RoboDK station: kr30 cnc 070119 curve 7 axis test 4.rdk

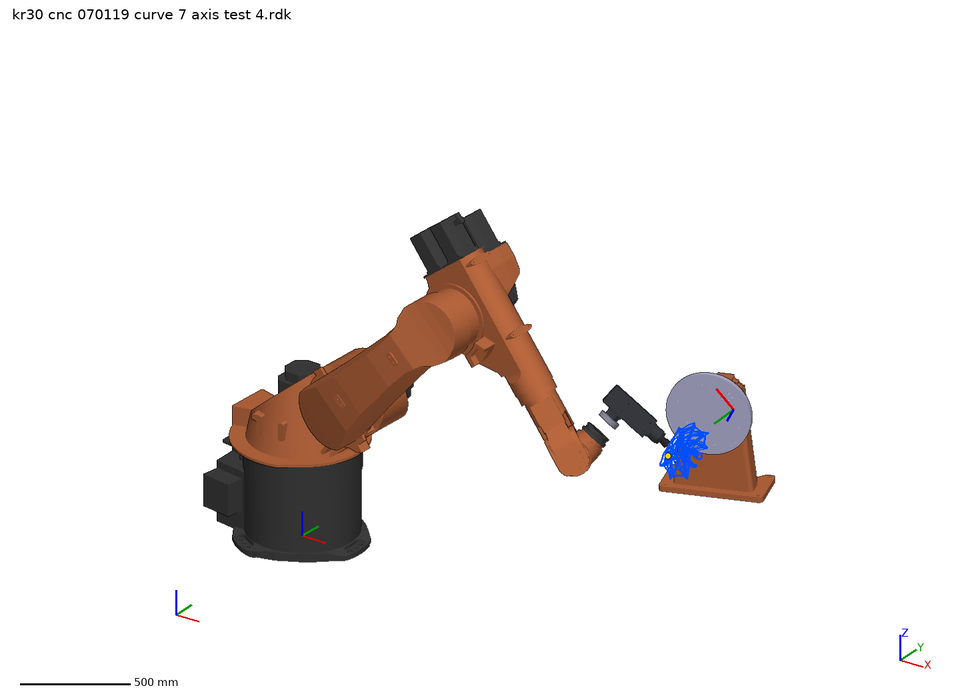
[picture v0: the station drawn from its stored meshes, robots at their saved joint values, targets as dots, program paths as lines]
Station kr30 cnc 070119 curve 7 axis test 4. Poses are relative to the parent item; angles as X-Y-Z fixed-axis rotations.
  - machining project Curve settings: C:/Temp/temp3/RhinoProject.stl | rotZ(0) | rotX(0)*rotY(0) | rotz(0) | onStart | onPathStart | onApproach | onPoint | onRetract | onFinish | onPathFinish | M_RunCode(%1)
  - frame KUKA KP1 MD250 Base at (0, 1000, 0) mm
    - robot KUKA KP1 MD250: 1 axes, payload 250 kg
        modified DH rows (alpha deg, a mm, theta deg, d mm): 0, 0, 0, 0
        base shift (1750, 1710, 820) mm, rotated rx 0 ry 90 rz -70 deg
        joint limits [-3600] to [3600]; home [0]; saved at [-138.652]
      - frame Reference Rhino at (0, -250, 250) mm
        - object RhinoPart at (0, 0, 0) mm
  - frame KUKA KR 30 HA Base at (0, 2000, 0) mm
    - robot KUKA KR 30 HA: 6 axes, payload 30 kg, reach 2033 mm, repeatability 0.05 mm, weight 665 kg
        modified DH rows (alpha deg, a mm, theta deg, d mm): 0, 0, 0, 815; -90, 350, 0, 0; 0, 850, -90, 0; -90, 145, 0, 820; 90, 0, 0, 0; -90, 0, 180, 170
        joint limits [-185, -135, -120, -350, -119, -350] to [185, 35, 158, 350, 119, 350]; home [0, -90, 90, 0, 0, 0]; saved at [2.992, -45.506, 98.07, 220.703, 109.004, -186.689]
      - tool 1/2" End Mill TCP, TCP at (337.71, -2.2, 160.57) mm, rotated rx 0 ry 90 rz 0 deg, size 415.8 x 102 x 153.6 mm
  - machining project RhinoPart Settings: rotZ(0) | rotX(90)*rotY(-155) | rotz(0) | onStart | onPathStart | onApproach | onPoint | onRetract | onFinish | onPathFinish | M_RunCode(%1)
  - program RhinoPart (1340 instructions, listed below)
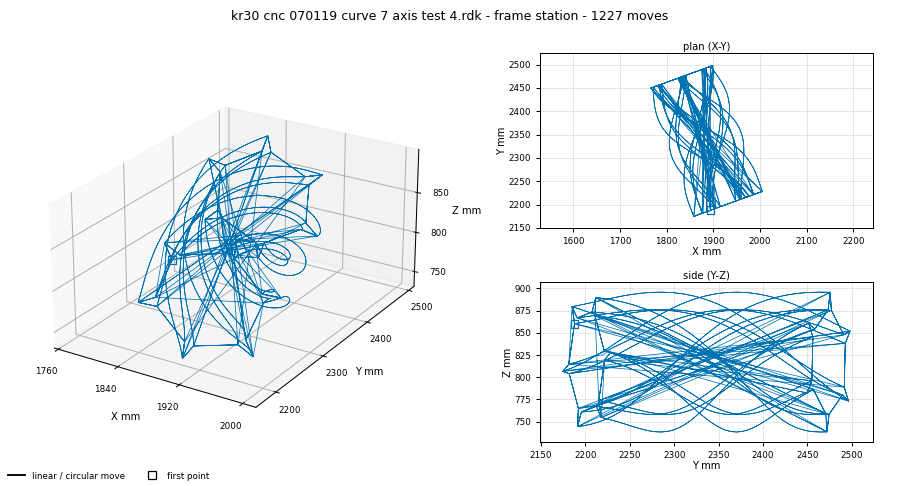
[picture p0: tool path of kr30 cnc 070119 curve 7 axis test 4.rdk in frame station, 1227 of 1227 moves have a stored position in this frame; points joined in program order, loops and branches not executed]

--- program RhinoPart (robot KUKA KR 30 HA) ---
  Set Ref.: Reference Rhino
  Set Tool: 1/2" End Mill TCP
  Show 1/2" End Mill TCP
  Set speed (1000.0 mm/s)
  MoveJ 1 to (58.93, 255.88, 290) mm, rotated rx -90 ry -25 rz 145.69 deg; joints [2.992, -45.858, 98.042, 220.619, 108.716, -186.951, -185.694]
  MoveL 2 to (58.93, 255.88, 290) mm, rotated rx -90 ry -25 rz 145.69 deg; joints [2.992, -45.858, 98.042, 220.619, 108.716, -186.951, -185.694]
  MoveL 3 to (58.93, 255.88, 290) mm, rotated rx -90 ry -25 rz 145.69 deg; joints [2.992, -45.858, 98.042, 220.619, 108.716, -186.951, -185.694]
  Set speed (60.0 mm/s)
  MoveL 4 to (37.11, 300.24, 290) mm, rotated rx -90 ry -25 rz -166.45 deg; joints [2.992, -46.004, 98.028, 220.584, 108.594, -187.061, -233.547]
  MoveL 5 to (-37.11, 208.63, 290) mm, rotated rx -90 ry -25 rz 8.11 deg; joints [2.992, -45.692, 98.056, 220.659, 108.852, -186.827, -408.107]
  Set speed (60.0 mm/s)
  MoveL 6 to (-58.93, 252.99, 290) mm, rotated rx -90 ry -25 rz -42.9 deg; joints [2.992, -45.848, 98.043, 220.621, 108.724, -186.944, -357.096]
  MoveL 7 to (21.11, 199.39, 290) mm, rotated rx -90 ry -25 rz 72.64 deg; joints [2.992, -45.658, 98.059, 220.667, 108.88, -186.802, -472.645]
  Set speed (60.0 mm/s)
  MoveL 8 to (34.79, 183.72, 290) mm, rotated rx -90 ry -25 rz 77.69 deg; joints [2.992, -46.56, 97.967, 220.451, 108.125, -187.483, -477.692]
  MoveL 9 to (21.11, 199.39, 290) mm, rotated rx -90 ry -25 rz 72.64 deg; joints [2.992, -45.658, 98.059, 220.667, 108.88, -186.802, -472.645]
  Set speed (60.0 mm/s)
  MoveL 10 to (-28.22, 202.67, 290) mm, rotated rx -90 ry -25 rz 19.2 deg; joints [2.992, -45.67, 98.058, 220.664, 108.87, -186.811, -419.196]
  MoveL 11 to (-43.85, 188.95, 290) mm, rotated rx -90 ry -25 rz 14.31 deg; joints [2.992, -46.574, 97.966, 220.447, 108.114, -187.494, -414.314]
  Set speed (60.0 mm/s)
  MoveL 12 to (-28.22, 202.67, 290) mm, rotated rx -90 ry -25 rz 19.2 deg; joints [2.992, -45.67, 98.058, 220.664, 108.87, -186.811, -419.196]
  MoveL 13 to (-43.85, 188.95, 290) mm, rotated rx -90 ry -25 rz 14.31 deg; joints [2.992, -46.574, 97.966, 220.447, 108.114, -187.494, -414.314]
  Set speed (60.0 mm/s)
  MoveL 14 to (-37.11, 208.63, 290) mm, rotated rx -90 ry -25 rz 8.11 deg; joints [2.992, -45.692, 98.056, 220.659, 108.852, -186.827, -408.107]
  MoveL 15 to (-78.63, 259.66, 290) mm, rotated rx -90 ry -25 rz -47.01 deg; joints [2.992, -46.754, 97.943, 220.404, 107.959, -187.632, -352.994]
  Set speed (60.0 mm/s)
  MoveL 16 to (-58.93, 252.99, 290) mm, rotated rx -90 ry -25 rz -42.9 deg; joints [2.992, -45.848, 98.043, 220.621, 108.724, -186.944, -357.096]
  MoveL 17 to (-78.63, 259.66, 290) mm, rotated rx -90 ry -25 rz -47.01 deg; joints [2.992, -46.754, 97.943, 220.404, 107.959, -187.632, -352.994]
  Set speed (60.0 mm/s)
  MoveL 18 to (-58.22, 263.67, 290) mm, rotated rx -90 ry -25 rz -53.21 deg; joints [2.992, -45.884, 98.039, 220.612, 108.694, -186.971, -346.787]
  MoveL 19 to (-30.72, 304.75, 290) mm, rotated rx -90 ry -25 rz -100.71 deg; joints [2.992, -46.018, 98.027, 220.58, 108.582, -187.072, -299.294]
  Set speed (60.0 mm/s)
  MoveL 20 to (-58.22, 263.67, 290) mm, rotated rx -90 ry -25 rz -53.21 deg; joints [2.992, -45.884, 98.039, 220.612, 108.694, -186.971, -346.787]
  MoveL 21 to (-30.72, 304.75, 290) mm, rotated rx -90 ry -25 rz -100.71 deg; joints [2.992, -46.018, 98.027, 220.58, 108.582, -187.072, -299.294]
  Set speed (60.0 mm/s)
  MoveL 22 to (-34.79, 325.15, 290) mm, rotated rx -90 ry -25 rz -105.16 deg; joints [2.992, -46.913, 97.922, 220.367, 107.822, -187.755, -294.84]
  MoveL 23 to (-21.11, 309.47, 290) mm, rotated rx -90 ry -25 rz -110.46 deg; joints [2.992, -46.033, 98.025, 220.576, 108.57, -187.083, -289.544]
  Set speed (60.0 mm/s)
  MoveL 24 to (-34.79, 325.15, 290) mm, rotated rx -90 ry -25 rz -105.16 deg; joints [2.992, -46.913, 97.922, 220.367, 107.822, -187.755, -294.84]
  MoveL 25 to (-21.11, 309.47, 290) mm, rotated rx -90 ry -25 rz -110.46 deg; joints [2.992, -46.033, 98.025, 220.576, 108.57, -187.083, -289.544]
  Set speed (60.0 mm/s)
  MoveL 26 to (28.22, 306.19, 290) mm, rotated rx -90 ry -25 rz -156.66 deg; joints [2.992, -46.023, 98.026, 220.579, 108.578, -187.075, -243.337]
  MoveL 27 to (43.85, 319.91, 290) mm, rotated rx -90 ry -25 rz -162.09 deg; joints [2.992, -46.901, 97.924, 220.37, 107.832, -187.745, -237.907]
  Set speed (60.0 mm/s)
  MoveL 28 to (28.22, 306.19, 290) mm, rotated rx -90 ry -25 rz -156.66 deg; joints [2.992, -46.023, 98.026, 220.579, 108.578, -187.075, -243.337]
  MoveL 29 to (43.85, 319.91, 290) mm, rotated rx -90 ry -25 rz -162.09 deg; joints [2.992, -46.901, 97.924, 220.37, 107.832, -187.745, -237.907]
  Set speed (60.0 mm/s)
  MoveL 30 to (37.11, 300.24, 290) mm, rotated rx -90 ry -25 rz -166.45 deg; joints [2.992, -46.004, 98.028, 220.584, 108.594, -187.061, -233.547]
  MoveL 31 to (78.63, 249.2, 290) mm, rotated rx -90 ry -25 rz 139.42 deg; joints [2.992, -46.728, 97.946, 220.411, 107.981, -187.612, -179.419]
  Set speed (60.0 mm/s)
  MoveL 32 to (58.93, 255.88, 290) mm, rotated rx -90 ry -25 rz 145.69 deg; joints [2.992, -45.858, 98.042, 220.619, 108.716, -186.951, -185.694]
  MoveL 33 to (78.63, 249.2, 290) mm, rotated rx -90 ry -25 rz 139.42 deg; joints [2.992, -46.728, 97.946, 220.411, 107.981, -187.612, -179.419]
  Set speed (60.0 mm/s)
  MoveL 34 to (58.22, 245.2, 290) mm, rotated rx -90 ry -25 rz 135.28 deg; joints [2.992, -45.821, 98.045, 220.627, 108.746, -186.924, -175.284]
  MoveL 35 to (30.72, 204.12, 290) mm, rotated rx -90 ry -25 rz 83.8 deg; joints [2.992, -45.676, 98.058, 220.663, 108.866, -186.815, -123.801]
  Set speed (60.0 mm/s)
  MoveL 36 to (58.22, 245.2, 290) mm, rotated rx -90 ry -25 rz 135.28 deg; joints [2.992, -45.821, 98.045, 220.627, 108.746, -186.924, -175.284]
  MoveL 37 to (30.72, 204.12, 290) mm, rotated rx -90 ry -25 rz 83.8 deg; joints [2.992, -45.676, 98.058, 220.663, 108.866, -186.815, -123.801]
  Set speed (60.0 mm/s)
  MoveL 38 to (34.79, 183.72, 290) mm, rotated rx -90 ry -25 rz 77.69 deg; joints [2.992, -46.56, 97.967, 220.451, 108.125, -187.483, -117.692]
  MoveL 39 to (-37.62, 299.82, 0) mm, rotated rx -90 ry -25 rz -92.94 deg; joints [-7.468, -50.311, 106.419, 214.538, 108.079, -179.325, 52.939]
  Set speed (60.0 mm/s)
  MoveL 40 to (10.16, 312.5, 0) mm, rotated rx -90 ry -25 rz -139.23 deg; joints [-7.468, -50.355, 106.415, 214.529, 108.039, -179.354, 99.233]
  MoveL 41 to (-37.62, 299.82, 0) mm, rotated rx -90 ry -25 rz -92.94 deg; joints [-7.468, -50.311, 106.419, 214.538, 108.079, -179.325, 52.939]
  Set speed (60.0 mm/s)
  MoveL 42 to (-55.59, 310.29, 0) mm, rotated rx -90 ry -25 rz -87.32 deg; joints [-7.468, -51.259, 106.317, 214.349, 107.213, -179.948, 47.319]
  MoveL 43 to (-45.21, 292.27, 0) mm, rotated rx -90 ry -25 rz -83.07 deg; joints [-7.468, -50.285, 106.421, 214.543, 108.102, -179.308, 43.073]
  Set speed (60.0 mm/s)
  MoveL 44 to (-55.59, 310.29, 0) mm, rotated rx -90 ry -25 rz -87.32 deg; joints [-7.468, -51.259, 106.317, 214.349, 107.213, -179.948, 47.319]
  MoveL 45 to (-45.21, 292.27, 0) mm, rotated rx -90 ry -25 rz -83.07 deg; joints [-7.468, -50.285, 106.421, 214.543, 108.102, -179.308, 43.073]
  Set speed (60.0 mm/s)
  MoveL 46 to (-58.12, 244.54, 0) mm, rotated rx -90 ry -25 rz -34.64 deg; joints [-7.468, -50.113, 106.436, 214.578, 108.256, -179.196, -5.364]
  MoveL 47 to (-76.17, 234.21, 0) mm, rotated rx -90 ry -25 rz -28.29 deg; joints [-7.468, -51.057, 106.341, 214.389, 107.4, -179.814, -11.709]
  Set speed (60.0 mm/s)
  MoveL 48 to (-58.12, 244.54, 0) mm, rotated rx -90 ry -25 rz -34.64 deg; joints [-7.468, -50.113, 106.436, 214.578, 108.256, -179.196, -5.364]
  MoveL 49 to (-76.17, 234.21, 0) mm, rotated rx -90 ry -25 rz -28.29 deg; joints [-7.468, -51.057, 106.341, 214.389, 107.4, -179.814, -11.709]
  Set speed (60.0 mm/s)
  MoveL 50 to (-55.37, 234.2, 0) mm, rotated rx -90 ry -25 rz -24.07 deg; joints [-7.468, -50.074, 106.439, 214.586, 108.291, -179.171, -15.929]
  MoveL 51 to (-20.49, 199.16, 0) mm, rotated rx -90 ry -25 rz 28.05 deg; joints [-7.468, -49.938, 106.45, 214.613, 108.412, -179.083, -68.047]
  Set speed (60.0 mm/s)
  MoveL 52 to (-55.37, 234.2, 0) mm, rotated rx -90 ry -25 rz -24.07 deg; joints [-7.468, -50.074, 106.439, 214.586, 108.291, -179.171, -15.929]
  MoveL 53 to (-20.49, 199.16, 0) mm, rotated rx -90 ry -25 rz 28.05 deg; joints [-7.468, -49.938, 106.45, 214.613, 108.412, -179.083, -68.047]
  Set speed (60.0 mm/s)
  MoveL 54 to (-20.57, 178.36, 0) mm, rotated rx -90 ry -25 rz 33.98 deg; joints [-7.468, -50.9, 106.359, 214.42, 107.545, -179.71, -73.977]
  MoveL 55 to (-10.16, 196.36, 0) mm, rotated rx -90 ry -25 rz 39.27 deg; joints [-7.468, -49.927, 106.451, 214.616, 108.422, -179.076, -79.273]
  Set speed (60.0 mm/s)
  MoveL 56 to (-20.57, 178.36, 0) mm, rotated rx -90 ry -25 rz 33.98 deg; joints [-7.468, -50.9, 106.359, 214.42, 107.545, -179.71, -73.977]
  MoveL 57 to (-10.16, 196.36, 0) mm, rotated rx -90 ry -25 rz 39.27 deg; joints [-7.468, -49.927, 106.451, 214.616, 108.422, -179.076, -79.273]
  Set speed (60.0 mm/s)
  MoveL 58 to (37.62, 209.05, 0) mm, rotated rx -90 ry -25 rz 92.57 deg; joints [-7.468, -49.977, 106.447, 214.605, 108.377, -179.109, -132.574]
  MoveL 59 to (55.59, 198.58, 0) mm, rotated rx -90 ry -25 rz 97.23 deg; joints [-7.468, -50.957, 106.353, 214.408, 107.492, -179.748, -137.234]
  Set speed (60.0 mm/s)
  MoveL 60 to (37.62, 209.05, 0) mm, rotated rx -90 ry -25 rz 92.57 deg; joints [-7.468, -49.977, 106.447, 214.605, 108.377, -179.109, -132.574]
  MoveL 61 to (55.59, 198.58, 0) mm, rotated rx -90 ry -25 rz 97.23 deg; joints [-7.468, -50.957, 106.353, 214.408, 107.492, -179.748, -137.234]
  Set speed (60.0 mm/s)
  MoveL 62 to (45.21, 216.6, 0) mm, rotated rx -90 ry -25 rz 103.54 deg; joints [-7.468, -50.007, 106.445, 214.599, 108.351, -179.128, -143.543]
  MoveL 63 to (58.12, 264.32, 0) mm, rotated rx -90 ry -25 rz 153.85 deg; joints [-7.468, -50.186, 106.43, 214.563, 108.191, -179.243, -193.845]
  Set speed (60.0 mm/s)
  MoveL 64 to (45.21, 216.6, 0) mm, rotated rx -90 ry -25 rz 103.54 deg; joints [-7.468, -50.007, 106.445, 214.599, 108.351, -179.128, -143.543]
  MoveL 65 to (58.12, 264.32, 0) mm, rotated rx -90 ry -25 rz 153.85 deg; joints [-7.468, -50.186, 106.43, 214.563, 108.191, -179.243, -193.845]
  Set speed (60.0 mm/s)
  MoveL 66 to (76.17, 274.65, 0) mm, rotated rx -90 ry -25 rz 157.93 deg; joints [-7.468, -51.166, 106.328, 214.367, 107.299, -179.886, -197.935]
  MoveL 67 to (55.37, 274.67, 0) mm, rotated rx -90 ry -25 rz 164.01 deg; joints [-7.468, -50.223, 106.427, 214.556, 108.158, -179.268, -204.014]
  Set speed (60.0 mm/s)
  MoveL 68 to (76.17, 274.65, 0) mm, rotated rx -90 ry -25 rz 157.93 deg; joints [-7.468, -51.166, 106.328, 214.367, 107.299, -179.886, -197.935]
  MoveL 69 to (55.37, 274.67, 0) mm, rotated rx -90 ry -25 rz 164.01 deg; joints [-7.468, -50.223, 106.427, 214.556, 108.158, -179.268, -204.014]
  Set speed (60.0 mm/s)
  MoveL 70 to (20.49, 309.71, 0) mm, rotated rx -90 ry -25 rz -148.94 deg; joints [-7.468, -50.346, 106.416, 214.531, 108.048, -179.347, -251.057]
  MoveL 71 to (20.57, 330.51, 0) mm, rotated rx -90 ry -25 rz -144.34 deg; joints [-7.468, -51.311, 106.31, 214.338, 107.164, -179.983, -255.665]
  Set speed (60.0 mm/s)
  MoveL 72 to (20.49, 309.71, 0) mm, rotated rx -90 ry -25 rz -148.94 deg; joints [-7.468, -50.346, 106.416, 214.531, 108.048, -179.347, -251.057]
  MoveL 73 to (20.57, 330.51, 0) mm, rotated rx -90 ry -25 rz -144.34 deg; joints [-7.468, -51.311, 106.31, 214.338, 107.164, -179.983, -255.665]
  Set speed (60.0 mm/s)
  MoveL 74 to (10.16, 312.5, 0) mm, rotated rx -90 ry -25 rz -139.23 deg; joints [-7.468, -50.355, 106.415, 214.529, 108.039, -179.354, -260.767]
  MoveL 75 to (-37.62, 299.82, 0) mm, rotated rx -90 ry -25 rz -92.94 deg; joints [-7.468, -50.311, 106.419, 214.538, 108.079, -179.325, -307.061]
  Set speed (60.0 mm/s)
  MoveL 76 to (-40.85, 296.93, 10) mm, rotated rx -90 ry -25 rz -88.96 deg; joints [-7.088, -50.198, 106.219, 214.78, 108.128, -179.56, -311.039]
  MoveL 77 to (-44.15, 293.5, 20) mm, rotated rx -90 ry -25 rz -84.58 deg; joints [-6.709, -50.079, 106.012, 215.02, 108.177, -179.796, -315.425]
  MoveL 78 to (-47.39, 289.5, 30) mm, rotated rx -90 ry -25 rz -79.81 deg; joints [-6.332, -49.955, 105.8, 215.259, 108.227, -180.032, -320.19]
  MoveL 79 to (-50.45, 284.92, 40) mm, rotated rx -90 ry -25 rz -74.69 deg; joints [-5.956, -49.826, 105.582, 215.496, 108.277, -180.268, -325.308]
  MoveL 80 to (-53.21, 279.8, 50) mm, rotated rx -90 ry -25 rz -69.25 deg; joints [-5.581, -49.692, 105.357, 215.732, 108.326, -180.504, -330.751]
  MoveL 81 to (-55.55, 274.16, 60) mm, rotated rx -90 ry -25 rz -63.51 deg; joints [-5.207, -49.552, 105.127, 215.966, 108.376, -180.74, -336.493]
  MoveL 82 to (-57.35, 268.08, 70) mm, rotated rx -90 ry -25 rz -57.49 deg; joints [-4.834, -49.408, 104.89, 216.198, 108.425, -180.977, -342.507]
  MoveL 83 to (-58.51, 261.62, 80) mm, rotated rx -90 ry -25 rz -51.24 deg; joints [-4.463, -49.259, 104.647, 216.429, 108.474, -181.215, -348.765]
  MoveL 84 to (-58.95, 254.91, 90) mm, rotated rx -90 ry -25 rz -44.76 deg; joints [-4.093, -49.106, 104.398, 216.657, 108.522, -181.454, -355.24]
  MoveL 85 to (-58.6, 248.05, 100) mm, rotated rx -90 ry -25 rz -38.1 deg; joints [-3.725, -48.95, 104.143, 216.884, 108.569, -181.693, -361.902]
  MoveL 86 to (-57.44, 241.19, 110) mm, rotated rx -90 ry -25 rz -31.28 deg; joints [-3.358, -48.79, 103.881, 217.108, 108.614, -181.935, -368.721]
  MoveL 87 to (-55.46, 234.45, 120) mm, rotated rx -90 ry -25 rz -24.34 deg; joints [-2.992, -48.627, 103.613, 217.33, 108.658, -182.178, -375.664]
  MoveL 88 to (-52.68, 227.97, 130) mm, rotated rx -90 ry -25 rz -17.3 deg; joints [-2.628, -48.462, 103.339, 217.55, 108.698, -182.423, -382.696]
  MoveL 89 to (-49.15, 221.88, 140) mm, rotated rx -90 ry -25 rz -10.22 deg; joints [-2.265, -48.294, 103.059, 217.767, 108.736, -182.671, -389.78]
  MoveL 90 to (-44.94, 216.28, 150) mm, rotated rx -90 ry -25 rz -3.12 deg; joints [-1.904, -48.126, 102.771, 217.981, 108.771, -182.922, -396.877]
  MoveL 91 to (-40.17, 211.29, 160) mm, rotated rx -90 ry -25 rz 3.94 deg; joints [-1.544, -47.956, 102.478, 218.192, 108.802, -183.176, -403.944]
  MoveL 92 to (-34.94, 206.95, 170) mm, rotated rx -90 ry -25 rz 10.94 deg; joints [-1.185, -47.786, 102.178, 218.401, 108.829, -183.434, -410.939]
  MoveL 93 to (-29.38, 203.32, 180) mm, rotated rx -90 ry -25 rz 17.81 deg; joints [-0.828, -47.615, 101.871, 218.606, 108.852, -183.696, -417.814]
  MoveL 94 to (-23.62, 200.42, 190) mm, rotated rx -90 ry -25 rz 24.52 deg; joints [-0.473, -47.444, 101.557, 218.809, 108.871, -183.961, -424.525]
  MoveL 95 to (-17.8, 198.23, 200) mm, rotated rx -90 ry -25 rz 31.02 deg; joints [-0.119, -47.272, 101.237, 219.008, 108.886, -184.23, -431.023]
  MoveL 96 to (-12.04, 196.73, 210) mm, rotated rx -90 ry -25 rz 37.26 deg; joints [0.233, -47.1, 100.911, 219.204, 108.897, -184.503, -437.262]
  MoveL 97 to (-6.46, 195.84, 220) mm, rotated rx -90 ry -25 rz 43.2 deg; joints [0.584, -46.927, 100.577, 219.397, 108.905, -184.78, -443.197]
  MoveL 98 to (-1.16, 195.49, 230) mm, rotated rx -90 ry -25 rz 48.78 deg; joints [0.933, -46.752, 100.237, 219.587, 108.909, -185.06, -448.782]
  MoveL 99 to (3.78, 195.6, 240) mm, rotated rx -90 ry -25 rz 53.97 deg; joints [1.28, -46.576, 99.891, 219.774, 108.91, -185.344, -453.974]
  MoveL 100 to (8.28, 196.07, 250) mm, rotated rx -90 ry -25 rz 58.73 deg; joints [1.626, -46.398, 99.538, 219.958, 108.908, -185.631, -458.733]
  MoveL 101 to (12.3, 196.78, 260) mm, rotated rx -90 ry -25 rz 63.02 deg; joints [1.97, -46.218, 99.178, 220.139, 108.904, -185.92, -463.017]
  MoveL 102 to (15.8, 197.64, 270) mm, rotated rx -90 ry -25 rz 66.79 deg; joints [2.312, -46.035, 98.812, 220.318, 108.898, -186.212, -466.788]
  MoveL 103 to (18.74, 198.54, 280) mm, rotated rx -90 ry -25 rz 70.01 deg; joints [2.653, -45.848, 98.439, 220.494, 108.89, -186.506, -470.01]
  MoveL 104 to (21.11, 199.39, 290) mm, rotated rx -90 ry -25 rz 72.64 deg; joints [2.992, -45.658, 98.059, 220.667, 108.88, -186.802, -472.645]
  MoveL 105 to (10.16, 312.5, 0) mm, rotated rx -90 ry -25 rz -139.23 deg; joints [-7.468, -50.355, 106.415, 214.529, 108.039, -179.354, -620.767]
  Set speed (60.0 mm/s)
  MoveL 106 to (-37.62, 299.82, 0) mm, rotated rx -90 ry -25 rz -92.94 deg; joints [-7.468, -50.311, 106.419, 214.538, 108.079, -179.325, -667.061]
  MoveL 107 to (-28.22, 202.67, 290) mm, rotated rx -90 ry -25 rz 19.2 deg; joints [2.992, -45.67, 98.058, 220.664, 108.87, -186.811, -779.196]
  Set speed (60.0 mm/s)
  MoveL 108 to (21.11, 199.39, 290) mm, rotated rx -90 ry -25 rz 72.64 deg; joints [2.992, -45.658, 98.059, 220.667, 108.88, -186.802, -832.645]
  MoveL 109 to (-28.22, 202.67, 290) mm, rotated rx -90 ry -25 rz 19.2 deg; joints [2.992, -45.67, 98.058, 220.664, 108.87, -186.811, -779.196]
  Set speed (60.0 mm/s)
  MoveL 110 to (-30.4, 203.93, 280) mm, rotated rx -90 ry -25 rz 16.58 deg; joints [2.653, -45.868, 98.437, 220.489, 108.873, -186.521, -776.579]
  MoveL 111 to (-33, 205.58, 270) mm, rotated rx -90 ry -25 rz 13.39 deg; joints [2.312, -46.064, 98.809, 220.311, 108.874, -186.234, -773.391]
  MoveL 112 to (-35.92, 207.69, 260) mm, rotated rx -90 ry -25 rz 9.67 deg; joints [1.97, -46.258, 99.175, 220.13, 108.871, -185.95, -769.674]
  MoveL 113 to (-39.07, 210.28, 250) mm, rotated rx -90 ry -25 rz 5.47 deg; joints [1.626, -46.451, 99.533, 219.946, 108.865, -185.669, -765.473]
  MoveL 114 to (-42.34, 213.41, 240) mm, rotated rx -90 ry -25 rz 0.83 deg; joints [1.28, -46.642, 99.885, 219.758, 108.855, -185.392, -760.831]
  MoveL 115 to (-45.62, 217.1, 230) mm, rotated rx -90 ry -25 rz -4.21 deg; joints [0.933, -46.832, 100.231, 219.568, 108.842, -185.119, -755.794]
  MoveL 116 to (-48.8, 221.36, 220) mm, rotated rx -90 ry -25 rz -9.59 deg; joints [0.584, -47.021, 100.57, 219.375, 108.826, -184.849, -750.406]
  MoveL 117 to (-51.74, 226.19, 210) mm, rotated rx -90 ry -25 rz -15.29 deg; joints [0.233, -47.209, 100.902, 219.178, 108.806, -184.582, -744.713]
  MoveL 118 to (-54.33, 231.55, 200) mm, rotated rx -90 ry -25 rz -21.24 deg; joints [-0.119, -47.395, 101.227, 218.979, 108.783, -184.319, -738.758]
  MoveL 119 to (-56.44, 237.4, 190) mm, rotated rx -90 ry -25 rz -27.41 deg; joints [-0.473, -47.58, 101.546, 218.777, 108.756, -184.059, -732.587]
  MoveL 120 to (-57.96, 243.66, 180) mm, rotated rx -90 ry -25 rz -33.76 deg; joints [-0.828, -47.763, 101.858, 218.572, 108.727, -183.801, -726.24]
  MoveL 121 to (-58.8, 250.25, 170) mm, rotated rx -90 ry -25 rz -40.24 deg; joints [-1.185, -47.944, 102.164, 218.365, 108.694, -183.547, -719.76]
  MoveL 122 to (-58.89, 257.04, 160) mm, rotated rx -90 ry -25 rz -46.82 deg; joints [-1.544, -48.123, 102.464, 218.154, 108.66, -183.294, -713.183]
  MoveL 123 to (-58.18, 263.92, 150) mm, rotated rx -90 ry -25 rz -53.45 deg; joints [-1.904, -48.298, 102.757, 217.942, 108.623, -183.043, -706.549]
  MoveL 124 to (-56.65, 270.74, 140) mm, rotated rx -90 ry -25 rz -60.11 deg; joints [-2.265, -48.47, 103.043, 217.727, 108.585, -182.794, -699.89]
  MoveL 125 to (-54.3, 277.38, 130) mm, rotated rx -90 ry -25 rz -66.76 deg; joints [-2.628, -48.638, 103.324, 217.51, 108.546, -182.546, -693.241]
  MoveL 126 to (-51.17, 283.7, 120) mm, rotated rx -90 ry -25 rz -73.37 deg; joints [-2.992, -48.802, 103.598, 217.291, 108.506, -182.299, -686.632]
  MoveL 127 to (-47.33, 289.58, 110) mm, rotated rx -90 ry -25 rz -79.91 deg; joints [-3.358, -48.961, 103.866, 217.07, 108.466, -182.053, -680.094]
  MoveL 128 to (-42.85, 294.92, 100) mm, rotated rx -90 ry -25 rz -86.35 deg; joints [-3.725, -49.114, 104.128, 216.848, 108.426, -181.807, -673.654]
  MoveL 129 to (-37.86, 299.62, 90) mm, rotated rx -90 ry -25 rz -92.66 deg; joints [-4.093, -49.263, 104.384, 216.623, 108.386, -181.561, -667.341]
  MoveL 130 to (-32.46, 303.64, 80) mm, rotated rx -90 ry -25 rz -98.82 deg; joints [-4.463, -49.406, 104.634, 216.397, 108.346, -181.315, -661.181]
  MoveL 131 to (-26.8, 306.94, 70) mm, rotated rx -90 ry -25 rz -104.8 deg; joints [-4.834, -49.543, 104.878, 216.169, 108.307, -181.069, -655.202]
  MoveL 132 to (-21, 309.52, 60) mm, rotated rx -90 ry -25 rz -110.57 deg; joints [-5.207, -49.675, 105.115, 215.94, 108.268, -180.823, -649.431]
  MoveL 133 to (-15.19, 311.39, 50) mm, rotated rx -90 ry -25 rz -116.1 deg; joints [-5.581, -49.801, 105.347, 215.709, 108.23, -180.577, -643.896]
  MoveL 134 to (-9.5, 312.61, 40) mm, rotated rx -90 ry -25 rz -121.38 deg; joints [-5.956, -49.921, 105.573, 215.476, 108.192, -180.331, -638.624]
  MoveL 135 to (-4.03, 313.25, 30) mm, rotated rx -90 ry -25 rz -126.35 deg; joints [-6.332, -50.037, 105.793, 215.242, 108.154, -180.086, -633.645]
  MoveL 136 to (1.12, 313.37, 20) mm, rotated rx -90 ry -25 rz -131.01 deg; joints [-6.709, -50.147, 106.006, 215.006, 108.116, -179.841, -628.989]
  MoveL 137 to (5.87, 313.09, 10) mm, rotated rx -90 ry -25 rz -135.31 deg; joints [-7.088, -50.253, 106.214, 214.768, 108.078, -179.597, -624.685]
  MoveL 138 to (10.16, 312.5, 0) mm, rotated rx -90 ry -25 rz -139.23 deg; joints [-7.468, -50.355, 106.415, 214.529, 108.039, -179.354, -620.767]
  MoveL 139 to (-37.62, 299.82, 0) mm, rotated rx -90 ry -25 rz -92.94 deg; joints [-7.468, -50.311, 106.419, 214.538, 108.079, -179.325, -667.061]
  Set speed (60.0 mm/s)
  MoveL 140 to (-40.85, 296.93, 10) mm, rotated rx -90 ry -25 rz -88.96 deg; joints [-7.088, -50.198, 106.219, 214.78, 108.128, -179.56, -671.039]
  MoveL 141 to (-44.15, 293.5, 20) mm, rotated rx -90 ry -25 rz -84.58 deg; joints [-6.709, -50.079, 106.012, 215.02, 108.177, -179.796, -675.425]
  MoveL 142 to (-47.39, 289.5, 30) mm, rotated rx -90 ry -25 rz -79.81 deg; joints [-6.332, -49.955, 105.8, 215.259, 108.227, -180.032, -680.19]
  MoveL 143 to (-50.45, 284.92, 40) mm, rotated rx -90 ry -25 rz -74.69 deg; joints [-5.956, -49.826, 105.582, 215.496, 108.277, -180.268, -685.308]
  MoveL 144 to (-53.21, 279.8, 50) mm, rotated rx -90 ry -25 rz -69.25 deg; joints [-5.581, -49.692, 105.357, 215.732, 108.326, -180.504, -690.751]
  MoveL 145 to (-55.55, 274.16, 60) mm, rotated rx -90 ry -25 rz -63.51 deg; joints [-5.207, -49.552, 105.127, 215.966, 108.376, -180.74, -696.493]
  MoveL 146 to (-57.35, 268.08, 70) mm, rotated rx -90 ry -25 rz -57.49 deg; joints [-4.834, -49.408, 104.89, 216.198, 108.425, -180.977, -702.507]
  MoveL 147 to (-58.51, 261.62, 80) mm, rotated rx -90 ry -25 rz -51.24 deg; joints [-4.463, -49.259, 104.647, 216.429, 108.474, -181.215, -708.765]
  MoveL 148 to (-58.95, 254.91, 90) mm, rotated rx -90 ry -25 rz -44.76 deg; joints [-4.093, -49.106, 104.398, 216.657, 108.522, -181.454, -715.24]
  MoveL 149 to (-58.6, 248.05, 100) mm, rotated rx -90 ry -25 rz -38.1 deg; joints [-3.725, -48.95, 104.143, 216.884, 108.569, -181.693, -721.902]
  MoveL 150 to (-57.44, 241.19, 110) mm, rotated rx -90 ry -25 rz -31.28 deg; joints [-3.358, -48.79, 103.881, 217.108, 108.614, -181.935, -728.721]
  MoveL 151 to (-55.46, 234.45, 120) mm, rotated rx -90 ry -25 rz -24.34 deg; joints [-2.992, -48.627, 103.613, 217.33, 108.658, -182.178, -735.664]
  MoveL 152 to (-52.68, 227.97, 130) mm, rotated rx -90 ry -25 rz -17.3 deg; joints [-2.628, -48.462, 103.339, 217.55, 108.698, -182.423, -742.696]
  MoveL 153 to (-49.15, 221.88, 140) mm, rotated rx -90 ry -25 rz -10.22 deg; joints [-2.265, -48.294, 103.059, 217.767, 108.736, -182.671, -749.78]
  MoveL 154 to (-44.94, 216.28, 150) mm, rotated rx -90 ry -25 rz -3.12 deg; joints [-1.904, -48.126, 102.771, 217.981, 108.771, -182.922, -756.877]
  MoveL 155 to (-40.17, 211.29, 160) mm, rotated rx -90 ry -25 rz 3.94 deg; joints [-1.544, -47.956, 102.478, 218.192, 108.802, -183.176, -763.944]
  MoveL 156 to (-34.94, 206.95, 170) mm, rotated rx -90 ry -25 rz 10.94 deg; joints [-1.185, -47.786, 102.178, 218.401, 108.829, -183.434, -770.939]
  MoveL 157 to (-29.38, 203.32, 180) mm, rotated rx -90 ry -25 rz 17.81 deg; joints [-0.828, -47.615, 101.871, 218.606, 108.852, -183.696, -777.814]
  MoveL 158 to (-23.62, 200.42, 190) mm, rotated rx -90 ry -25 rz 24.52 deg; joints [-0.473, -47.444, 101.557, 218.809, 108.871, -183.961, -784.525]
  MoveL 159 to (-17.8, 198.23, 200) mm, rotated rx -90 ry -25 rz 31.02 deg; joints [-0.119, -47.272, 101.237, 219.008, 108.886, -184.23, -791.023]
  MoveL 160 to (-12.04, 196.73, 210) mm, rotated rx -90 ry -25 rz 37.26 deg; joints [0.233, -47.1, 100.911, 219.204, 108.897, -184.503, -797.262]
  MoveL 161 to (-6.46, 195.84, 220) mm, rotated rx -90 ry -25 rz 43.2 deg; joints [0.584, -46.927, 100.577, 219.397, 108.905, -184.78, -803.197]
  MoveL 162 to (-1.16, 195.49, 230) mm, rotated rx -90 ry -25 rz 48.78 deg; joints [0.933, -46.752, 100.237, 219.587, 108.909, -185.06, -808.782]
  MoveL 163 to (3.78, 195.6, 240) mm, rotated rx -90 ry -25 rz 53.97 deg; joints [1.28, -46.576, 99.891, 219.774, 108.91, -185.344, -813.974]
  MoveL 164 to (8.28, 196.07, 250) mm, rotated rx -90 ry -25 rz 58.73 deg; joints [1.626, -46.398, 99.538, 219.958, 108.908, -185.631, -818.733]
  MoveL 165 to (12.3, 196.78, 260) mm, rotated rx -90 ry -25 rz 63.02 deg; joints [1.97, -46.218, 99.178, 220.139, 108.904, -185.92, -823.017]
  MoveL 166 to (15.8, 197.64, 270) mm, rotated rx -90 ry -25 rz 66.79 deg; joints [2.312, -46.035, 98.812, 220.318, 108.898, -186.212, -826.788]
  MoveL 167 to (18.74, 198.54, 280) mm, rotated rx -90 ry -25 rz 70.01 deg; joints [2.653, -45.848, 98.439, 220.494, 108.89, -186.506, -830.01]
  MoveL 168 to (21.11, 199.39, 290) mm, rotated rx -90 ry -25 rz 72.64 deg; joints [2.992, -45.658, 98.059, 220.667, 108.88, -186.802, -832.645]
  MoveL 169 to (34.79, 183.72, 290) mm, rotated rx -90 ry -25 rz 77.69 deg; joints [2.992, -46.56, 97.967, 220.451, 108.125, -187.483, -837.692]
  Set speed (60.0 mm/s)
  MoveL 170 to (21.11, 199.39, 290) mm, rotated rx -90 ry -25 rz 72.64 deg; joints [2.992, -45.658, 98.059, 220.667, 108.88, -186.802, -832.645]
  MoveL 171 to (-55.59, 310.29, 0) mm, rotated rx -90 ry -25 rz -87.32 deg; joints [-7.468, -51.259, 106.317, 214.349, 107.213, -179.948, -672.681]
  Set speed (60.0 mm/s)
  MoveL 172 to (-37.62, 299.82, 0) mm, rotated rx -90 ry -25 rz -92.94 deg; joints [-7.468, -50.311, 106.419, 214.538, 108.079, -179.325, -667.061]
  MoveL 173 to (34.79, 183.72, 290) mm, rotated rx -90 ry -25 rz 77.69 deg; joints [2.992, -46.56, 97.967, 220.451, 108.125, -187.483, -837.692]
  Set speed (60.0 mm/s)
  MoveL 174 to (31.73, 182.3, 280) mm, rotated rx -90 ry -25 rz 75.11 deg; joints [2.653, -46.752, 98.347, 220.278, 108.131, -187.186, -835.112]
  MoveL 175 to (27.92, 180.74, 270) mm, rotated rx -90 ry -25 rz 71.96 deg; joints [2.312, -46.941, 98.72, 220.102, 108.136, -186.891, -831.958]
  MoveL 176 to (23.38, 179.17, 260) mm, rotated rx -90 ry -25 rz 68.27 deg; joints [1.97, -47.126, 99.087, 219.924, 108.139, -186.598, -828.265]
  MoveL 177 to (18.11, 177.74, 250) mm, rotated rx -90 ry -25 rz 64.07 deg; joints [1.626, -47.308, 99.447, 219.743, 108.14, -186.307, -824.071]
  MoveL 178 to (12.17, 176.57, 240) mm, rotated rx -90 ry -25 rz 59.41 deg; joints [1.28, -47.487, 99.8, 219.56, 108.139, -186.019, -819.412]
  MoveL 179 to (5.61, 175.83, 230) mm, rotated rx -90 ry -25 rz 54.33 deg; joints [0.933, -47.665, 100.147, 219.373, 108.135, -185.733, -814.325]
  MoveL 180 to (-1.49, 175.64, 220) mm, rotated rx -90 ry -25 rz 48.85 deg; joints [0.584, -47.84, 100.487, 219.184, 108.128, -185.451, -808.851]
  MoveL 181 to (-9.03, 176.15, 210) mm, rotated rx -90 ry -25 rz 43.03 deg; joints [0.233, -48.014, 100.82, 218.992, 108.118, -185.172, -803.03]
  MoveL 182 to (-16.88, 177.46, 200) mm, rotated rx -90 ry -25 rz 36.9 deg; joints [-0.119, -48.187, 101.147, 218.797, 108.104, -184.896, -796.902]
  MoveL 183 to (-24.89, 179.66, 190) mm, rotated rx -90 ry -25 rz 30.51 deg; joints [-0.473, -48.36, 101.467, 218.598, 108.086, -184.624, -790.512]
  MoveL 184 to (-32.91, 182.83, 180) mm, rotated rx -90 ry -25 rz 23.9 deg; joints [-0.828, -48.531, 101.78, 218.397, 108.064, -184.356, -783.901]
  MoveL 185 to (-40.75, 186.98, 170) mm, rotated rx -90 ry -25 rz 17.11 deg; joints [-1.185, -48.702, 102.087, 218.193, 108.039, -184.092, -777.113]
  MoveL 186 to (-48.24, 192.12, 160) mm, rotated rx -90 ry -25 rz 10.19 deg; joints [-1.544, -48.873, 102.387, 217.985, 108.009, -183.831, -770.193]
  MoveL 187 to (-55.2, 198.19, 150) mm, rotated rx -90 ry -25 rz 3.18 deg; joints [-1.904, -49.043, 102.68, 217.775, 107.975, -183.574, -763.183]
  MoveL 188 to (-61.48, 205.13, 140) mm, rotated rx -90 ry -25 rz -3.87 deg; joints [-2.265, -49.212, 102.967, 217.562, 107.937, -183.321, -756.127]
  MoveL 189 to (-66.92, 212.81, 130) mm, rotated rx -90 ry -25 rz -10.94 deg; joints [-2.628, -49.38, 103.247, 217.346, 107.896, -183.07, -749.064]
  MoveL 190 to (-71.41, 221.1, 120) mm, rotated rx -90 ry -25 rz -17.96 deg; joints [-2.992, -49.546, 103.52, 217.128, 107.851, -182.823, -742.035]
  MoveL 191 to (-74.87, 229.83, 110) mm, rotated rx -90 ry -25 rz -24.92 deg; joints [-3.358, -49.71, 103.787, 216.907, 107.804, -182.577, -735.078]
  MoveL 192 to (-77.24, 238.83, 100) mm, rotated rx -90 ry -25 rz -31.77 deg; joints [-3.725, -49.872, 104.048, 216.684, 107.755, -182.334, -728.229]
  MoveL 193 to (-78.53, 247.91, 90) mm, rotated rx -90 ry -25 rz -38.48 deg; joints [-4.093, -50.03, 104.302, 216.459, 107.704, -182.093, -721.522]
  MoveL 194 to (-78.77, 256.9, 80) mm, rotated rx -90 ry -25 rz -45.01 deg; joints [-4.463, -50.185, 104.551, 216.231, 107.651, -181.852, -714.991]
  MoveL 195 to (-78, 265.63, 70) mm, rotated rx -90 ry -25 rz -51.33 deg; joints [-4.834, -50.336, 104.793, 216.002, 107.597, -181.613, -708.666]
  MoveL 196 to (-76.35, 273.96, 60) mm, rotated rx -90 ry -25 rz -57.42 deg; joints [-5.207, -50.483, 105.028, 215.77, 107.542, -181.374, -702.579]
  MoveL 197 to (-73.92, 281.75, 50) mm, rotated rx -90 ry -25 rz -63.24 deg; joints [-5.581, -50.625, 105.258, 215.538, 107.487, -181.136, -696.759]
  MoveL 198 to (-70.87, 288.9, 40) mm, rotated rx -90 ry -25 rz -68.76 deg; joints [-5.956, -50.762, 105.482, 215.303, 107.432, -180.898, -691.235]
  MoveL 199 to (-67.34, 295.36, 30) mm, rotated rx -90 ry -25 rz -73.96 deg; joints [-6.332, -50.894, 105.7, 215.067, 107.377, -180.661, -686.036]
  MoveL 200 to (-63.51, 301.08, 20) mm, rotated rx -90 ry -25 rz -78.81 deg; joints [-6.709, -51.021, 105.911, 214.829, 107.322, -180.423, -681.192]
  MoveL 201 to (-59.54, 306.05, 10) mm, rotated rx -90 ry -25 rz -83.27 deg; joints [-7.088, -51.143, 106.117, 214.59, 107.267, -180.186, -676.73]
  MoveL 202 to (-55.59, 310.29, 0) mm, rotated rx -90 ry -25 rz -87.32 deg; joints [-7.468, -51.259, 106.317, 214.349, 107.213, -179.948, -672.681]
  MoveL 203 to (34.79, 183.72, 290) mm, rotated rx -90 ry -25 rz 77.69 deg; joints [2.992, -46.56, 97.967, 220.451, 108.125, -187.483, -837.692]
  Set speed (60.0 mm/s)
  MoveL 204 to (30.72, 204.12, 290) mm, rotated rx -90 ry -25 rz 83.8 deg; joints [2.992, -45.676, 98.058, 220.663, 108.866, -186.815, -843.801]
  MoveL 205 to (-55.59, 310.29, 0) mm, rotated rx -90 ry -25 rz -87.32 deg; joints [-7.468, -51.259, 106.317, 214.349, 107.213, -179.948, -672.681]
  Set speed (60.0 mm/s)
  MoveL 206 to (-45.21, 292.27, 0) mm, rotated rx -90 ry -25 rz -83.07 deg; joints [-7.468, -50.285, 106.421, 214.543, 108.102, -179.308, -676.927]
  MoveL 207 to (-55.59, 310.29, 0) mm, rotated rx -90 ry -25 rz -87.32 deg; joints [-7.468, -51.259, 106.317, 214.349, 107.213, -179.948, -672.681]
  Set speed (60.0 mm/s)
  MoveL 208 to (-59.54, 306.05, 10) mm, rotated rx -90 ry -25 rz -83.27 deg; joints [-7.088, -51.143, 106.117, 214.59, 107.267, -180.186, -676.73]
  MoveL 209 to (-63.51, 301.08, 20) mm, rotated rx -90 ry -25 rz -78.81 deg; joints [-6.709, -51.021, 105.911, 214.829, 107.322, -180.423, -681.192]
  MoveL 210 to (-67.34, 295.36, 30) mm, rotated rx -90 ry -25 rz -73.96 deg; joints [-6.332, -50.894, 105.7, 215.067, 107.377, -180.661, -686.036]
  MoveL 211 to (-70.87, 288.9, 40) mm, rotated rx -90 ry -25 rz -68.76 deg; joints [-5.956, -50.762, 105.482, 215.303, 107.432, -180.898, -691.235]
  MoveL 212 to (-73.92, 281.75, 50) mm, rotated rx -90 ry -25 rz -63.24 deg; joints [-5.581, -50.625, 105.258, 215.538, 107.487, -181.136, -696.759]
  MoveL 213 to (-76.35, 273.96, 60) mm, rotated rx -90 ry -25 rz -57.42 deg; joints [-5.207, -50.483, 105.028, 215.77, 107.542, -181.374, -702.579]
  MoveL 214 to (-78, 265.63, 70) mm, rotated rx -90 ry -25 rz -51.33 deg; joints [-4.834, -50.336, 104.793, 216.002, 107.597, -181.613, -708.666]
  MoveL 215 to (-78.77, 256.9, 80) mm, rotated rx -90 ry -25 rz -45.01 deg; joints [-4.463, -50.185, 104.551, 216.231, 107.651, -181.852, -714.991]
  MoveL 216 to (-78.53, 247.91, 90) mm, rotated rx -90 ry -25 rz -38.48 deg; joints [-4.093, -50.03, 104.302, 216.459, 107.704, -182.093, -721.522]
  MoveL 217 to (-77.24, 238.83, 100) mm, rotated rx -90 ry -25 rz -31.77 deg; joints [-3.725, -49.872, 104.048, 216.684, 107.755, -182.334, -728.229]
  MoveL 218 to (-74.87, 229.83, 110) mm, rotated rx -90 ry -25 rz -24.92 deg; joints [-3.358, -49.71, 103.787, 216.907, 107.804, -182.577, -735.078]
  MoveL 219 to (-71.41, 221.1, 120) mm, rotated rx -90 ry -25 rz -17.96 deg; joints [-2.992, -49.546, 103.52, 217.128, 107.851, -182.823, -742.035]
  MoveL 220 to (-66.92, 212.81, 130) mm, rotated rx -90 ry -25 rz -10.94 deg; joints [-2.628, -49.38, 103.247, 217.346, 107.896, -183.07, -749.064]
  MoveL 221 to (-61.48, 205.13, 140) mm, rotated rx -90 ry -25 rz -3.87 deg; joints [-2.265, -49.212, 102.967, 217.562, 107.937, -183.321, -756.127]
  MoveL 222 to (-55.2, 198.19, 150) mm, rotated rx -90 ry -25 rz 3.18 deg; joints [-1.904, -49.043, 102.68, 217.775, 107.975, -183.574, -763.183]
  MoveL 223 to (-48.24, 192.12, 160) mm, rotated rx -90 ry -25 rz 10.19 deg; joints [-1.544, -48.873, 102.387, 217.985, 108.009, -183.831, -770.193]
  MoveL 224 to (-40.75, 186.98, 170) mm, rotated rx -90 ry -25 rz 17.11 deg; joints [-1.185, -48.702, 102.087, 218.193, 108.039, -184.092, -777.113]
  MoveL 225 to (-32.91, 182.83, 180) mm, rotated rx -90 ry -25 rz 23.9 deg; joints [-0.828, -48.531, 101.78, 218.397, 108.064, -184.356, -783.901]
  MoveL 226 to (-24.89, 179.66, 190) mm, rotated rx -90 ry -25 rz 30.51 deg; joints [-0.473, -48.36, 101.467, 218.598, 108.086, -184.624, -790.512]
  MoveL 227 to (-16.88, 177.46, 200) mm, rotated rx -90 ry -25 rz 36.9 deg; joints [-0.119, -48.187, 101.147, 218.797, 108.104, -184.896, -796.902]
  MoveL 228 to (-9.03, 176.15, 210) mm, rotated rx -90 ry -25 rz 43.03 deg; joints [0.233, -48.014, 100.82, 218.992, 108.118, -185.172, -803.03]
  MoveL 229 to (-1.49, 175.64, 220) mm, rotated rx -90 ry -25 rz 48.85 deg; joints [0.584, -47.84, 100.487, 219.184, 108.128, -185.451, -808.851]
  MoveL 230 to (5.61, 175.83, 230) mm, rotated rx -90 ry -25 rz 54.33 deg; joints [0.933, -47.665, 100.147, 219.373, 108.135, -185.733, -814.325]
  MoveL 231 to (12.17, 176.57, 240) mm, rotated rx -90 ry -25 rz 59.41 deg; joints [1.28, -47.487, 99.8, 219.56, 108.139, -186.019, -819.412]
  MoveL 232 to (18.11, 177.74, 250) mm, rotated rx -90 ry -25 rz 64.07 deg; joints [1.626, -47.308, 99.447, 219.743, 108.14, -186.307, -824.071]
  MoveL 233 to (23.38, 179.17, 260) mm, rotated rx -90 ry -25 rz 68.27 deg; joints [1.97, -47.126, 99.087, 219.924, 108.139, -186.598, -828.265]
  MoveL 234 to (27.92, 180.74, 270) mm, rotated rx -90 ry -25 rz 71.96 deg; joints [2.312, -46.941, 98.72, 220.102, 108.136, -186.891, -831.958]
  MoveL 235 to (31.73, 182.3, 280) mm, rotated rx -90 ry -25 rz 75.11 deg; joints [2.653, -46.752, 98.347, 220.278, 108.131, -187.186, -835.112]
  MoveL 236 to (34.79, 183.72, 290) mm, rotated rx -90 ry -25 rz 77.69 deg; joints [2.992, -46.56, 97.967, 220.451, 108.125, -187.483, -837.692]
  MoveL 237 to (30.72, 204.12, 290) mm, rotated rx -90 ry -25 rz 83.8 deg; joints [2.992, -45.676, 98.058, 220.663, 108.866, -186.815, -843.801]
  Set speed (60.0 mm/s)
  MoveL 238 to (28.54, 202.85, 280) mm, rotated rx -90 ry -25 rz 81.18 deg; joints [2.653, -45.864, 98.438, 220.49, 108.877, -186.518, -841.184]
  MoveL 239 to (25.81, 201.43, 270) mm, rotated rx -90 ry -25 rz 77.98 deg; joints [2.312, -46.049, 98.811, 220.314, 108.886, -186.222, -837.983]
  MoveL 240 to (22.53, 199.96, 260) mm, rotated rx -90 ry -25 rz 74.23 deg; joints [1.97, -46.229, 99.177, 220.136, 108.895, -185.929, -834.232]
  MoveL 241 to (18.7, 198.53, 250) mm, rotated rx -90 ry -25 rz 69.97 deg; joints [1.626, -46.407, 99.537, 219.956, 108.901, -185.637, -829.967]
  MoveL 242 to (14.35, 197.26, 240) mm, rotated rx -90 ry -25 rz 65.22 deg; joints [1.28, -46.582, 99.89, 219.772, 108.905, -185.349, -825.225]
  MoveL 243 to (9.52, 196.26, 230) mm, rotated rx -90 ry -25 rz 60.04 deg; joints [0.933, -46.755, 100.237, 219.586, 108.907, -185.063, -820.042]
  MoveL 244 to (4.24, 195.64, 220) mm, rotated rx -90 ry -25 rz 54.46 deg; joints [0.584, -46.926, 100.577, 219.397, 108.906, -184.78, -814.46]
  MoveL 245 to (-1.41, 195.5, 210) mm, rotated rx -90 ry -25 rz 48.52 deg; joints [0.233, -47.095, 100.911, 219.205, 108.901, -184.5, -808.518]
  MoveL 246 to (-7.35, 195.94, 200) mm, rotated rx -90 ry -25 rz 42.26 deg; joints [-0.119, -47.264, 101.238, 219.01, 108.893, -184.224, -802.261]
  MoveL 247 to (-13.47, 197.04, 190) mm, rotated rx -90 ry -25 rz 35.73 deg; joints [-0.473, -47.431, 101.558, 218.812, 108.882, -183.952, -795.734]
  MoveL 248 to (-19.65, 198.85, 180) mm, rotated rx -90 ry -25 rz 28.98 deg; joints [-0.828, -47.598, 101.872, 218.61, 108.866, -183.684, -788.982]
  MoveL 249 to (-25.78, 201.42, 170) mm, rotated rx -90 ry -25 rz 22.05 deg; joints [-1.185, -47.765, 102.179, 218.406, 108.847, -183.419, -782.053]
  MoveL 250 to (-31.7, 204.73, 160) mm, rotated rx -90 ry -25 rz 14.99 deg; joints [-1.544, -47.932, 102.48, 218.198, 108.823, -183.159, -774.993]
  MoveL 251 to (-37.3, 208.79, 150) mm, rotated rx -90 ry -25 rz 7.85 deg; joints [-1.904, -48.098, 102.774, 217.987, 108.795, -182.902, -767.85]
  MoveL 252 to (-42.45, 213.53, 140) mm, rotated rx -90 ry -25 rz 0.67 deg; joints [-2.265, -48.263, 103.061, 217.774, 108.763, -182.649, -760.67]
  MoveL 253 to (-47.02, 218.88, 130) mm, rotated rx -90 ry -25 rz -6.5 deg; joints [-2.628, -48.428, 103.342, 217.557, 108.727, -182.399, -753.496]
  MoveL 254 to (-50.93, 224.75, 120) mm, rotated rx -90 ry -25 rz -13.63 deg; joints [-2.992, -48.591, 103.616, 217.338, 108.689, -182.153, -746.37]
  MoveL 255 to (-54.1, 231.02, 110) mm, rotated rx -90 ry -25 rz -20.67 deg; joints [-3.358, -48.752, 103.884, 217.116, 108.647, -181.909, -739.332]
  MoveL 256 to (-56.49, 237.56, 100) mm, rotated rx -90 ry -25 rz -27.58 deg; joints [-3.725, -48.911, 104.146, 216.892, 108.602, -181.667, -732.418]
  MoveL 257 to (-58.06, 244.24, 90) mm, rotated rx -90 ry -25 rz -34.34 deg; joints [-4.093, -49.068, 104.401, 216.666, 108.556, -181.427, -725.663]
  MoveL 258 to (-58.85, 250.92, 80) mm, rotated rx -90 ry -25 rz -40.9 deg; joints [-4.463, -49.221, 104.65, 216.437, 108.508, -181.189, -719.1]
  MoveL 259 to (-58.87, 257.48, 70) mm, rotated rx -90 ry -25 rz -47.24 deg; joints [-4.834, -49.37, 104.893, 216.206, 108.459, -180.952, -712.759]
  MoveL 260 to (-58.2, 263.79, 60) mm, rotated rx -90 ry -25 rz -53.33 deg; joints [-5.207, -49.515, 105.13, 215.974, 108.409, -180.716, -706.668]
  MoveL 261 to (-56.92, 269.76, 50) mm, rotated rx -90 ry -25 rz -59.14 deg; joints [-5.581, -49.656, 105.36, 215.739, 108.358, -180.48, -700.857]
  MoveL 262 to (-55.13, 275.3, 40) mm, rotated rx -90 ry -25 rz -64.65 deg; joints [-5.956, -49.792, 105.585, 215.503, 108.307, -180.245, -695.351]
  MoveL 263 to (-52.95, 280.35, 30) mm, rotated rx -90 ry -25 rz -69.82 deg; joints [-6.332, -49.923, 105.803, 215.266, 108.256, -180.01, -690.178]
  MoveL 264 to (-50.48, 284.87, 20) mm, rotated rx -90 ry -25 rz -74.63 deg; joints [-6.709, -50.049, 106.015, 215.026, 108.204, -179.776, -685.365]
  MoveL 265 to (-47.86, 288.84, 10) mm, rotated rx -90 ry -25 rz -79.06 deg; joints [-7.088, -50.169, 106.221, 214.785, 108.153, -179.542, -680.939]
  MoveL 266 to (-45.21, 292.27, 0) mm, rotated rx -90 ry -25 rz -83.07 deg; joints [-7.468, -50.285, 106.421, 214.543, 108.102, -179.308, -676.927]
  MoveL 267 to (30.72, 204.12, 290) mm, rotated rx -90 ry -25 rz 83.8 deg; joints [2.992, -45.676, 98.058, 220.663, 108.866, -186.815, -843.801]
  Set speed (60.0 mm/s)
  MoveL 268 to (58.22, 245.2, 290) mm, rotated rx -90 ry -25 rz 135.28 deg; joints [2.992, -45.821, 98.045, 220.627, 108.746, -186.924, -895.284]
  MoveL 269 to (-45.21, 292.27, 0) mm, rotated rx -90 ry -25 rz -83.07 deg; joints [-7.468, -50.285, 106.421, 214.543, 108.102, -179.308, -1036.927]
  Set speed (60.0 mm/s)
  MoveL 270 to (-58.12, 244.54, 0) mm, rotated rx -90 ry -25 rz -34.64 deg; joints [-7.468, -50.113, 106.436, 214.578, 108.256, -179.196, -1085.364]
  MoveL 271 to (-45.21, 292.27, 0) mm, rotated rx -90 ry -25 rz -83.07 deg; joints [-7.468, -50.285, 106.421, 214.543, 108.102, -179.308, -1036.927]
  Set speed (60.0 mm/s)
  MoveL 272 to (-47.86, 288.84, 10) mm, rotated rx -90 ry -25 rz -79.06 deg; joints [-7.088, -50.169, 106.221, 214.785, 108.153, -179.542, -1040.939]
  MoveL 273 to (-50.48, 284.87, 20) mm, rotated rx -90 ry -25 rz -74.63 deg; joints [-6.709, -50.049, 106.015, 215.026, 108.204, -179.776, -1045.365]
  MoveL 274 to (-52.95, 280.35, 30) mm, rotated rx -90 ry -25 rz -69.82 deg; joints [-6.332, -49.923, 105.803, 215.266, 108.256, -180.01, -1050.178]
  MoveL 275 to (-55.13, 275.3, 40) mm, rotated rx -90 ry -25 rz -64.65 deg; joints [-5.956, -49.792, 105.585, 215.503, 108.307, -180.245, -1055.351]
  MoveL 276 to (-56.92, 269.76, 50) mm, rotated rx -90 ry -25 rz -59.14 deg; joints [-5.581, -49.656, 105.36, 215.739, 108.358, -180.48, -1060.857]
  MoveL 277 to (-58.2, 263.79, 60) mm, rotated rx -90 ry -25 rz -53.33 deg; joints [-5.207, -49.515, 105.13, 215.974, 108.409, -180.716, -1066.668]
  MoveL 278 to (-58.87, 257.48, 70) mm, rotated rx -90 ry -25 rz -47.24 deg; joints [-4.834, -49.37, 104.893, 216.206, 108.459, -180.952, -1072.759]
  MoveL 279 to (-58.85, 250.92, 80) mm, rotated rx -90 ry -25 rz -40.9 deg; joints [-4.463, -49.221, 104.65, 216.437, 108.508, -181.189, -1079.1]
  MoveL 280 to (-58.06, 244.24, 90) mm, rotated rx -90 ry -25 rz -34.34 deg; joints [-4.093, -49.068, 104.401, 216.666, 108.556, -181.427, -1085.663]
  MoveL 281 to (-56.49, 237.56, 100) mm, rotated rx -90 ry -25 rz -27.58 deg; joints [-3.725, -48.911, 104.146, 216.892, 108.602, -181.667, -1092.418]
  MoveL 282 to (-54.1, 231.02, 110) mm, rotated rx -90 ry -25 rz -20.67 deg; joints [-3.358, -48.752, 103.884, 217.116, 108.647, -181.909, -1099.332]
  MoveL 283 to (-50.93, 224.75, 120) mm, rotated rx -90 ry -25 rz -13.63 deg; joints [-2.992, -48.591, 103.616, 217.338, 108.689, -182.153, -1106.37]
  MoveL 284 to (-47.02, 218.88, 130) mm, rotated rx -90 ry -25 rz -6.5 deg; joints [-2.628, -48.428, 103.342, 217.557, 108.727, -182.399, -1113.496]
  MoveL 285 to (-42.45, 213.53, 140) mm, rotated rx -90 ry -25 rz 0.67 deg; joints [-2.265, -48.263, 103.061, 217.774, 108.763, -182.649, -1120.67]
  MoveL 286 to (-37.3, 208.79, 150) mm, rotated rx -90 ry -25 rz 7.85 deg; joints [-1.904, -48.098, 102.774, 217.987, 108.795, -182.902, -1127.85]
  MoveL 287 to (-31.7, 204.73, 160) mm, rotated rx -90 ry -25 rz 14.99 deg; joints [-1.544, -47.932, 102.48, 218.198, 108.823, -183.159, -1134.993]
  MoveL 288 to (-25.78, 201.42, 170) mm, rotated rx -90 ry -25 rz 22.05 deg; joints [-1.185, -47.765, 102.179, 218.406, 108.847, -183.419, -1142.053]
  MoveL 289 to (-19.65, 198.85, 180) mm, rotated rx -90 ry -25 rz 28.98 deg; joints [-0.828, -47.598, 101.872, 218.61, 108.866, -183.684, -1148.982]
  MoveL 290 to (-13.47, 197.04, 190) mm, rotated rx -90 ry -25 rz 35.73 deg; joints [-0.473, -47.431, 101.558, 218.812, 108.882, -183.952, -1155.734]
  MoveL 291 to (-7.35, 195.94, 200) mm, rotated rx -90 ry -25 rz 42.26 deg; joints [-0.119, -47.264, 101.238, 219.01, 108.893, -184.224, -1162.261]
  MoveL 292 to (-1.41, 195.5, 210) mm, rotated rx -90 ry -25 rz 48.52 deg; joints [0.233, -47.095, 100.911, 219.205, 108.901, -184.5, -1168.518]
  MoveL 293 to (4.24, 195.64, 220) mm, rotated rx -90 ry -25 rz 54.46 deg; joints [0.584, -46.926, 100.577, 219.397, 108.906, -184.78, -1174.46]
  MoveL 294 to (9.52, 196.26, 230) mm, rotated rx -90 ry -25 rz 60.04 deg; joints [0.933, -46.755, 100.237, 219.586, 108.907, -185.063, -1180.042]
  MoveL 295 to (14.35, 197.26, 240) mm, rotated rx -90 ry -25 rz 65.22 deg; joints [1.28, -46.582, 99.89, 219.772, 108.905, -185.349, -1185.225]
  MoveL 296 to (18.7, 198.53, 250) mm, rotated rx -90 ry -25 rz 69.97 deg; joints [1.626, -46.407, 99.537, 219.956, 108.901, -185.637, -1189.967]
  MoveL 297 to (22.53, 199.96, 260) mm, rotated rx -90 ry -25 rz 74.23 deg; joints [1.97, -46.229, 99.177, 220.136, 108.895, -185.929, -1194.232]
  MoveL 298 to (25.81, 201.43, 270) mm, rotated rx -90 ry -25 rz 77.98 deg; joints [2.312, -46.049, 98.811, 220.314, 108.886, -186.222, -1197.983]
  MoveL 299 to (28.54, 202.85, 280) mm, rotated rx -90 ry -25 rz 81.18 deg; joints [2.653, -45.864, 98.438, 220.49, 108.877, -186.518, -1201.184]
  MoveL 300 to (30.72, 204.12, 290) mm, rotated rx -90 ry -25 rz 83.8 deg; joints [2.992, -45.676, 98.058, 220.663, 108.866, -186.815, -1203.801]
  MoveL 301 to (58.22, 245.2, 290) mm, rotated rx -90 ry -25 rz 135.28 deg; joints [2.992, -45.821, 98.045, 220.627, 108.746, -186.924, -1255.284]
  Set speed (60.0 mm/s)
  MoveL 302 to (57.77, 242.72, 280) mm, rotated rx -90 ry -25 rz 132.81 deg; joints [2.653, -46.006, 98.425, 220.456, 108.759, -186.624, -1252.814]
  MoveL 303 to (57.08, 239.72, 270) mm, rotated rx -90 ry -25 rz 129.79 deg; joints [2.312, -46.186, 98.799, 220.282, 108.773, -186.324, -1249.788]
  MoveL 304 to (56.08, 236.26, 260) mm, rotated rx -90 ry -25 rz 126.23 deg; joints [1.97, -46.361, 99.166, 220.105, 108.786, -186.025, -1246.235]
  MoveL 305 to (54.69, 232.42, 250) mm, rotated rx -90 ry -25 rz 122.18 deg; joints [1.626, -46.53, 99.527, 219.927, 108.798, -185.728, -1242.184]
  MoveL 306 to (52.84, 228.29, 240) mm, rotated rx -90 ry -25 rz 117.66 deg; joints [1.28, -46.696, 99.881, 219.746, 108.81, -185.432, -1237.664]
  MoveL 307 to (50.46, 223.96, 230) mm, rotated rx -90 ry -25 rz 112.71 deg; joints [0.933, -46.857, 100.229, 219.562, 108.822, -185.137, -1232.705]
  MoveL 308 to (47.51, 219.54, 220) mm, rotated rx -90 ry -25 rz 107.34 deg; joints [0.584, -47.015, 100.57, 219.376, 108.831, -184.844, -1227.337]
  MoveL 309 to (43.95, 215.15, 210) mm, rotated rx -90 ry -25 rz 101.59 deg; joints [0.233, -47.169, 100.905, 219.188, 108.84, -184.553, -1221.59]
  MoveL 310 to (39.77, 210.92, 200) mm, rotated rx -90 ry -25 rz 95.5 deg; joints [-0.119, -47.32, 101.233, 218.997, 108.846, -184.265, -1215.499]
  MoveL 311 to (34.96, 206.97, 190) mm, rotated rx -90 ry -25 rz 89.1 deg; joints [-0.473, -47.469, 101.555, 218.803, 108.85, -183.979, -1209.096]
  MoveL 312 to (29.57, 203.44, 180) mm, rotated rx -90 ry -25 rz 82.42 deg; joints [-0.828, -47.616, 101.871, 218.606, 108.852, -183.696, -1202.421]
  MoveL 313 to (23.65, 200.44, 170) mm, rotated rx -90 ry -25 rz 75.51 deg; joints [-1.185, -47.761, 102.18, 218.406, 108.85, -183.417, -1195.511]
  MoveL 314 to (17.28, 198.07, 160) mm, rotated rx -90 ry -25 rz 68.41 deg; joints [-1.544, -47.906, 102.482, 218.204, 108.844, -183.141, -1188.409]
  MoveL 315 to (10.57, 196.44, 150) mm, rotated rx -90 ry -25 rz 61.16 deg; joints [-1.904, -48.051, 102.777, 217.998, 108.835, -182.869, -1181.159]
  MoveL 316 to (3.62, 195.59, 140) mm, rotated rx -90 ry -25 rz 53.81 deg; joints [-2.265, -48.195, 103.067, 217.789, 108.821, -182.601, -1173.808]
  MoveL 317 to (-3.42, 195.58, 130) mm, rotated rx -90 ry -25 rz 46.4 deg; joints [-2.628, -48.339, 103.349, 217.577, 108.803, -182.338, -1166.404]
  MoveL 318 to (-10.42, 196.41, 120) mm, rotated rx -90 ry -25 rz 38.99 deg; joints [-2.992, -48.483, 103.625, 217.362, 108.781, -182.078, -1158.993]
  MoveL 319 to (-17.25, 198.06, 110) mm, rotated rx -90 ry -25 rz 31.62 deg; joints [-3.358, -48.627, 103.895, 217.144, 108.754, -181.823, -1151.625]
  MoveL 320 to (-23.78, 200.49, 100) mm, rotated rx -90 ry -25 rz 24.35 deg; joints [-3.725, -48.771, 104.157, 216.923, 108.724, -181.571, -1144.346]
  MoveL 321 to (-29.89, 203.62, 90) mm, rotated rx -90 ry -25 rz 17.2 deg; joints [-4.093, -48.915, 104.414, 216.699, 108.689, -181.323, -1137.203]
  MoveL 322 to (-35.48, 207.36, 80) mm, rotated rx -90 ry -25 rz 10.24 deg; joints [-4.463, -49.058, 104.664, 216.472, 108.65, -181.078, -1130.238]
  MoveL 323 to (-40.49, 211.59, 70) mm, rotated rx -90 ry -25 rz 3.49 deg; joints [-4.834, -49.199, 104.907, 216.243, 108.608, -180.837, -1123.492]
  MoveL 324 to (-44.86, 216.19, 60) mm, rotated rx -90 ry -25 rz -3 deg; joints [-5.207, -49.339, 105.145, 216.011, 108.563, -180.597, -1117.004]
  MoveL 325 to (-48.58, 221.03, 50) mm, rotated rx -90 ry -25 rz -9.19 deg; joints [-5.581, -49.477, 105.375, 215.777, 108.516, -180.36, -1110.81]
  MoveL 326 to (-51.63, 225.99, 40) mm, rotated rx -90 ry -25 rz -15.06 deg; joints [-5.956, -49.611, 105.6, 215.541, 108.466, -180.125, -1104.943]
  MoveL 327 to (-54.06, 230.92, 30) mm, rotated rx -90 ry -25 rz -20.56 deg; joints [-6.332, -49.743, 105.818, 215.303, 108.415, -179.891, -1099.435]
  MoveL 328 to (-55.91, 235.73, 20) mm, rotated rx -90 ry -25 rz -25.68 deg; joints [-6.709, -49.87, 106.03, 215.063, 108.363, -179.659, -1094.317]
  MoveL 329 to (-57.23, 240.3, 10) mm, rotated rx -90 ry -25 rz -30.38 deg; joints [-7.088, -49.994, 106.236, 214.821, 108.31, -179.427, -1089.617]
  MoveL 330 to (-58.12, 244.54, 0) mm, rotated rx -90 ry -25 rz -34.64 deg; joints [-7.468, -50.113, 106.436, 214.578, 108.256, -179.196, -1085.364]
  MoveL 331 to (58.22, 245.2, 290) mm, rotated rx -90 ry -25 rz 135.28 deg; joints [2.992, -45.821, 98.045, 220.627, 108.746, -186.924, -1255.284]
  Set speed (60.0 mm/s)
  MoveL 332 to (78.63, 249.2, 290) mm, rotated rx -90 ry -25 rz 139.42 deg; joints [2.992, -46.728, 97.946, 220.411, 107.981, -187.612, -1259.419]
  MoveL 333 to (-58.12, 244.54, 0) mm, rotated rx -90 ry -25 rz -34.64 deg; joints [-7.468, -50.113, 106.436, 214.578, 108.256, -179.196, -1085.364]
  Set speed (60.0 mm/s)
  MoveL 334 to (-76.17, 234.21, 0) mm, rotated rx -90 ry -25 rz -28.29 deg; joints [-7.468, -51.057, 106.341, 214.389, 107.4, -179.814, -1091.709]
  MoveL 335 to (-58.12, 244.54, 0) mm, rotated rx -90 ry -25 rz -34.64 deg; joints [-7.468, -50.113, 106.436, 214.578, 108.256, -179.196, -1085.364]
  Set speed (60.0 mm/s)
  MoveL 336 to (-57.23, 240.3, 10) mm, rotated rx -90 ry -25 rz -30.38 deg; joints [-7.088, -49.994, 106.236, 214.821, 108.31, -179.427, -1089.617]
  MoveL 337 to (-55.91, 235.73, 20) mm, rotated rx -90 ry -25 rz -25.68 deg; joints [-6.709, -49.87, 106.03, 215.063, 108.363, -179.659, -1094.317]
  MoveL 338 to (-54.06, 230.92, 30) mm, rotated rx -90 ry -25 rz -20.56 deg; joints [-6.332, -49.743, 105.818, 215.303, 108.415, -179.891, -1099.435]
  MoveL 339 to (-51.63, 225.99, 40) mm, rotated rx -90 ry -25 rz -15.06 deg; joints [-5.956, -49.611, 105.6, 215.541, 108.466, -180.125, -1104.943]
  MoveL 340 to (-48.58, 221.03, 50) mm, rotated rx -90 ry -25 rz -9.19 deg; joints [-5.581, -49.477, 105.375, 215.777, 108.516, -180.36, -1110.81]
  MoveL 341 to (-44.86, 216.19, 60) mm, rotated rx -90 ry -25 rz -3 deg; joints [-5.207, -49.339, 105.145, 216.011, 108.563, -180.597, -1117.004]
  MoveL 342 to (-40.49, 211.59, 70) mm, rotated rx -90 ry -25 rz 3.49 deg; joints [-4.834, -49.199, 104.907, 216.243, 108.608, -180.837, -1123.492]
  MoveL 343 to (-35.48, 207.36, 80) mm, rotated rx -90 ry -25 rz 10.24 deg; joints [-4.463, -49.058, 104.664, 216.472, 108.65, -181.078, -1130.238]
  MoveL 344 to (-29.89, 203.62, 90) mm, rotated rx -90 ry -25 rz 17.2 deg; joints [-4.093, -48.915, 104.414, 216.699, 108.689, -181.323, -1137.203]
  MoveL 345 to (-23.78, 200.49, 100) mm, rotated rx -90 ry -25 rz 24.35 deg; joints [-3.725, -48.771, 104.157, 216.923, 108.724, -181.571, -1144.346]
  MoveL 346 to (-17.25, 198.06, 110) mm, rotated rx -90 ry -25 rz 31.62 deg; joints [-3.358, -48.627, 103.895, 217.144, 108.754, -181.823, -1151.625]
  MoveL 347 to (-10.42, 196.41, 120) mm, rotated rx -90 ry -25 rz 38.99 deg; joints [-2.992, -48.483, 103.625, 217.362, 108.781, -182.078, -1158.993]
  MoveL 348 to (-3.42, 195.58, 130) mm, rotated rx -90 ry -25 rz 46.4 deg; joints [-2.628, -48.339, 103.349, 217.577, 108.803, -182.338, -1166.404]
  MoveL 349 to (3.62, 195.59, 140) mm, rotated rx -90 ry -25 rz 53.81 deg; joints [-2.265, -48.195, 103.067, 217.789, 108.821, -182.601, -1173.808]
  MoveL 350 to (10.57, 196.44, 150) mm, rotated rx -90 ry -25 rz 61.16 deg; joints [-1.904, -48.051, 102.777, 217.998, 108.835, -182.869, -1181.159]
  MoveL 351 to (17.28, 198.07, 160) mm, rotated rx -90 ry -25 rz 68.41 deg; joints [-1.544, -47.906, 102.482, 218.204, 108.844, -183.141, -1188.409]
  MoveL 352 to (23.65, 200.44, 170) mm, rotated rx -90 ry -25 rz 75.51 deg; joints [-1.185, -47.761, 102.18, 218.406, 108.85, -183.417, -1195.511]
  MoveL 353 to (29.57, 203.44, 180) mm, rotated rx -90 ry -25 rz 82.42 deg; joints [-0.828, -47.616, 101.871, 218.606, 108.852, -183.696, -1202.421]
  MoveL 354 to (34.96, 206.97, 190) mm, rotated rx -90 ry -25 rz 89.1 deg; joints [-0.473, -47.469, 101.555, 218.803, 108.85, -183.979, -1209.096]
  MoveL 355 to (39.77, 210.92, 200) mm, rotated rx -90 ry -25 rz 95.5 deg; joints [-0.119, -47.32, 101.233, 218.997, 108.846, -184.265, -1215.499]
  MoveL 356 to (43.95, 215.15, 210) mm, rotated rx -90 ry -25 rz 101.59 deg; joints [0.233, -47.169, 100.905, 219.188, 108.84, -184.553, -1221.59]
  MoveL 357 to (47.51, 219.54, 220) mm, rotated rx -90 ry -25 rz 107.34 deg; joints [0.584, -47.015, 100.57, 219.376, 108.831, -184.844, -1227.337]
  MoveL 358 to (50.46, 223.96, 230) mm, rotated rx -90 ry -25 rz 112.71 deg; joints [0.933, -46.857, 100.229, 219.562, 108.822, -185.137, -1232.705]
  MoveL 359 to (52.84, 228.29, 240) mm, rotated rx -90 ry -25 rz 117.66 deg; joints [1.28, -46.696, 99.881, 219.746, 108.81, -185.432, -1237.664]
  MoveL 360 to (54.69, 232.42, 250) mm, rotated rx -90 ry -25 rz 122.18 deg; joints [1.626, -46.53, 99.527, 219.927, 108.798, -185.728, -1242.184]
  MoveL 361 to (56.08, 236.26, 260) mm, rotated rx -90 ry -25 rz 126.23 deg; joints [1.97, -46.361, 99.166, 220.105, 108.786, -186.025, -1246.235]
  MoveL 362 to (57.08, 239.72, 270) mm, rotated rx -90 ry -25 rz 129.79 deg; joints [2.312, -46.186, 98.799, 220.282, 108.773, -186.324, -1249.788]
  MoveL 363 to (57.77, 242.72, 280) mm, rotated rx -90 ry -25 rz 132.81 deg; joints [2.653, -46.006, 98.425, 220.456, 108.759, -186.624, -1252.814]
  MoveL 364 to (58.22, 245.2, 290) mm, rotated rx -90 ry -25 rz 135.28 deg; joints [2.992, -45.821, 98.045, 220.627, 108.746, -186.924, -1255.284]
  MoveL 365 to (78.63, 249.2, 290) mm, rotated rx -90 ry -25 rz 139.42 deg; joints [2.992, -46.728, 97.946, 220.411, 107.981, -187.612, -1259.419]
  Set speed (60.0 mm/s)
  MoveL 366 to (78.34, 245.85, 280) mm, rotated rx -90 ry -25 rz 136.96 deg; joints [2.653, -46.916, 98.327, 220.239, 107.991, -187.312, -1256.964]
  MoveL 367 to (77.78, 241.77, 270) mm, rotated rx -90 ry -25 rz 133.96 deg; joints [2.312, -47.099, 98.701, 220.065, 108, -187.012, -1253.959]
  MoveL 368 to (76.86, 237.05, 260) mm, rotated rx -90 ry -25 rz 130.43 deg; joints [1.97, -47.277, 99.068, 219.888, 108.009, -186.712, -1250.435]
  MoveL 369 to (75.48, 231.77, 250) mm, rotated rx -90 ry -25 rz 126.42 deg; joints [1.626, -47.45, 99.43, 219.71, 108.018, -186.414, -1246.422]
  MoveL 370 to (73.51, 226.04, 240) mm, rotated rx -90 ry -25 rz 121.95 deg; joints [1.28, -47.618, 99.784, 219.529, 108.026, -186.117, -1241.95]
  MoveL 371 to (70.88, 219.99, 230) mm, rotated rx -90 ry -25 rz 117.05 deg; joints [0.933, -47.782, 100.133, 219.346, 108.033, -185.821, -1237.052]
  MoveL 372 to (67.49, 213.75, 220) mm, rotated rx -90 ry -25 rz 111.76 deg; joints [0.584, -47.942, 100.475, 219.16, 108.039, -185.526, -1231.756]
  MoveL 373 to (63.28, 207.47, 210) mm, rotated rx -90 ry -25 rz 106.1 deg; joints [0.233, -48.099, 100.81, 218.972, 108.044, -185.234, -1226.097]
  MoveL 374 to (58.22, 201.33, 200) mm, rotated rx -90 ry -25 rz 100.11 deg; joints [-0.119, -48.252, 101.139, 218.782, 108.048, -184.944, -1220.107]
  MoveL 375 to (52.31, 195.49, 190) mm, rotated rx -90 ry -25 rz 93.82 deg; joints [-0.473, -48.403, 101.462, 218.589, 108.049, -184.656, -1213.819]
  MoveL 376 to (45.56, 190.13, 180) mm, rotated rx -90 ry -25 rz 87.27 deg; joints [-0.828, -48.551, 101.778, 218.393, 108.047, -184.371, -1207.271]
  MoveL 377 to (38.04, 185.42, 170) mm, rotated rx -90 ry -25 rz 80.5 deg; joints [-1.185, -48.698, 102.087, 218.194, 108.042, -184.089, -1200.5]
  MoveL 378 to (29.85, 181.5, 160) mm, rotated rx -90 ry -25 rz 73.54 deg; joints [-1.544, -48.844, 102.39, 217.992, 108.034, -183.81, -1193.545]
  MoveL 379 to (21.11, 178.51, 150) mm, rotated rx -90 ry -25 rz 66.45 deg; joints [-1.904, -48.989, 102.686, 217.787, 108.022, -183.536, -1186.447]
  MoveL 380 to (11.96, 176.54, 140) mm, rotated rx -90 ry -25 rz 59.25 deg; joints [-2.265, -49.133, 102.976, 217.58, 108.007, -183.265, -1179.249]
  MoveL 381 to (2.59, 175.67, 130) mm, rotated rx -90 ry -25 rz 51.99 deg; joints [-2.628, -49.278, 103.259, 217.369, 107.986, -182.998, -1171.995]
  MoveL 382 to (-6.83, 175.92, 120) mm, rotated rx -90 ry -25 rz 44.73 deg; joints [-2.992, -49.422, 103.535, 217.155, 107.962, -182.735, -1164.728]
  MoveL 383 to (-16.13, 177.3, 110) mm, rotated rx -90 ry -25 rz 37.49 deg; joints [-3.358, -49.566, 103.804, 216.938, 107.933, -182.476, -1157.494]
  MoveL 384 to (-25.11, 179.73, 100) mm, rotated rx -90 ry -25 rz 30.34 deg; joints [-3.725, -49.71, 104.067, 216.719, 107.9, -182.221, -1150.336]
  MoveL 385 to (-33.62, 183.16, 90) mm, rotated rx -90 ry -25 rz 23.3 deg; joints [-4.093, -49.853, 104.323, 216.496, 107.862, -181.969, -1143.298]
  MoveL 386 to (-41.52, 187.45, 80) mm, rotated rx -90 ry -25 rz 16.42 deg; joints [-4.463, -49.996, 104.573, 216.271, 107.821, -181.721, -1136.42]
  MoveL 387 to (-48.7, 192.48, 70) mm, rotated rx -90 ry -25 rz 9.74 deg; joints [-4.834, -50.138, 104.816, 216.043, 107.777, -181.476, -1129.745]
  MoveL 388 to (-55.08, 198.08, 60) mm, rotated rx -90 ry -25 rz 3.31 deg; joints [-5.207, -50.278, 105.053, 215.813, 107.729, -181.233, -1123.31]
  MoveL 389 to (-60.61, 204.07, 50) mm, rotated rx -90 ry -25 rz -2.85 deg; joints [-5.581, -50.415, 105.283, 215.581, 107.678, -180.993, -1117.152]
  MoveL 390 to (-65.29, 210.3, 40) mm, rotated rx -90 ry -25 rz -8.69 deg; joints [-5.956, -50.551, 105.507, 215.346, 107.625, -180.755, -1111.307]
  MoveL 391 to (-69.12, 216.58, 30) mm, rotated rx -90 ry -25 rz -14.19 deg; joints [-6.332, -50.683, 105.725, 215.11, 107.571, -180.518, -1105.808]
  MoveL 392 to (-72.16, 222.75, 20) mm, rotated rx -90 ry -25 rz -19.31 deg; joints [-6.709, -50.811, 105.937, 214.871, 107.515, -180.282, -1100.687]
  MoveL 393 to (-74.48, 228.68, 10) mm, rotated rx -90 ry -25 rz -24.02 deg; joints [-7.088, -50.936, 106.142, 214.631, 107.458, -180.048, -1095.978]
  MoveL 394 to (-76.17, 234.21, 0) mm, rotated rx -90 ry -25 rz -28.29 deg; joints [-7.468, -51.057, 106.341, 214.389, 107.4, -179.814, -1091.709]
  MoveL 395 to (78.63, 249.2, 290) mm, rotated rx -90 ry -25 rz 139.42 deg; joints [2.992, -46.728, 97.946, 220.411, 107.981, -187.612, -1259.419]
  Set speed (60.0 mm/s)
  MoveL 396 to (58.93, 255.88, 290) mm, rotated rx -90 ry -25 rz 145.69 deg; joints [2.992, -45.858, 98.042, 220.619, 108.716, -186.951, -1265.694]
  MoveL 397 to (-76.17, 234.21, 0) mm, rotated rx -90 ry -25 rz -28.29 deg; joints [-7.468, -51.057, 106.341, 214.389, 107.4, -179.814, -1091.709]
  Set speed (60.0 mm/s)
  MoveL 398 to (-55.37, 234.2, 0) mm, rotated rx -90 ry -25 rz -24.07 deg; joints [-7.468, -50.074, 106.439, 214.586, 108.291, -179.171, -1095.929]
  MoveL 399 to (-76.17, 234.21, 0) mm, rotated rx -90 ry -25 rz -28.29 deg; joints [-7.468, -51.057, 106.341, 214.389, 107.4, -179.814, -1091.709]
  Set speed (60.0 mm/s)
  MoveL 400 to (-74.48, 228.68, 10) mm, rotated rx -90 ry -25 rz -24.02 deg; joints [-7.088, -50.936, 106.142, 214.631, 107.458, -180.048, -1095.978]
  MoveL 401 to (-72.16, 222.75, 20) mm, rotated rx -90 ry -25 rz -19.31 deg; joints [-6.709, -50.811, 105.937, 214.871, 107.515, -180.282, -1100.687]
  MoveL 402 to (-69.12, 216.58, 30) mm, rotated rx -90 ry -25 rz -14.19 deg; joints [-6.332, -50.683, 105.725, 215.11, 107.571, -180.518, -1105.808]
  MoveL 403 to (-65.29, 210.3, 40) mm, rotated rx -90 ry -25 rz -8.69 deg; joints [-5.956, -50.551, 105.507, 215.346, 107.625, -180.755, -1111.307]
  MoveL 404 to (-60.61, 204.07, 50) mm, rotated rx -90 ry -25 rz -2.85 deg; joints [-5.581, -50.415, 105.283, 215.581, 107.678, -180.993, -1117.152]
  MoveL 405 to (-55.08, 198.08, 60) mm, rotated rx -90 ry -25 rz 3.31 deg; joints [-5.207, -50.278, 105.053, 215.813, 107.729, -181.233, -1123.31]
  MoveL 406 to (-48.7, 192.48, 70) mm, rotated rx -90 ry -25 rz 9.74 deg; joints [-4.834, -50.138, 104.816, 216.043, 107.777, -181.476, -1129.745]
  MoveL 407 to (-41.52, 187.45, 80) mm, rotated rx -90 ry -25 rz 16.42 deg; joints [-4.463, -49.996, 104.573, 216.271, 107.821, -181.721, -1136.42]
  MoveL 408 to (-33.62, 183.16, 90) mm, rotated rx -90 ry -25 rz 23.3 deg; joints [-4.093, -49.853, 104.323, 216.496, 107.862, -181.969, -1143.298]
  MoveL 409 to (-25.11, 179.73, 100) mm, rotated rx -90 ry -25 rz 30.34 deg; joints [-3.725, -49.71, 104.067, 216.719, 107.9, -182.221, -1150.336]
  MoveL 410 to (-16.13, 177.3, 110) mm, rotated rx -90 ry -25 rz 37.49 deg; joints [-3.358, -49.566, 103.804, 216.938, 107.933, -182.476, -1157.494]
  MoveL 411 to (-6.83, 175.92, 120) mm, rotated rx -90 ry -25 rz 44.73 deg; joints [-2.992, -49.422, 103.535, 217.155, 107.962, -182.735, -1164.728]
  MoveL 412 to (2.59, 175.67, 130) mm, rotated rx -90 ry -25 rz 51.99 deg; joints [-2.628, -49.278, 103.259, 217.369, 107.986, -182.998, -1171.995]
  MoveL 413 to (11.96, 176.54, 140) mm, rotated rx -90 ry -25 rz 59.25 deg; joints [-2.265, -49.133, 102.976, 217.58, 108.007, -183.265, -1179.249]
  MoveL 414 to (21.11, 178.51, 150) mm, rotated rx -90 ry -25 rz 66.45 deg; joints [-1.904, -48.989, 102.686, 217.787, 108.022, -183.536, -1186.447]
  MoveL 415 to (29.85, 181.5, 160) mm, rotated rx -90 ry -25 rz 73.54 deg; joints [-1.544, -48.844, 102.39, 217.992, 108.034, -183.81, -1193.545]
  MoveL 416 to (38.04, 185.42, 170) mm, rotated rx -90 ry -25 rz 80.5 deg; joints [-1.185, -48.698, 102.087, 218.194, 108.042, -184.089, -1200.5]
  MoveL 417 to (45.56, 190.13, 180) mm, rotated rx -90 ry -25 rz 87.27 deg; joints [-0.828, -48.551, 101.778, 218.393, 108.047, -184.371, -1207.271]
  MoveL 418 to (52.31, 195.49, 190) mm, rotated rx -90 ry -25 rz 93.82 deg; joints [-0.473, -48.403, 101.462, 218.589, 108.049, -184.656, -1213.819]
  MoveL 419 to (58.22, 201.33, 200) mm, rotated rx -90 ry -25 rz 100.11 deg; joints [-0.119, -48.252, 101.139, 218.782, 108.048, -184.944, -1220.107]
  MoveL 420 to (63.28, 207.47, 210) mm, rotated rx -90 ry -25 rz 106.1 deg; joints [0.233, -48.099, 100.81, 218.972, 108.044, -185.234, -1226.097]
  MoveL 421 to (67.49, 213.75, 220) mm, rotated rx -90 ry -25 rz 111.76 deg; joints [0.584, -47.942, 100.475, 219.16, 108.039, -185.526, -1231.756]
  MoveL 422 to (70.88, 219.99, 230) mm, rotated rx -90 ry -25 rz 117.05 deg; joints [0.933, -47.782, 100.133, 219.346, 108.033, -185.821, -1237.052]
  MoveL 423 to (73.51, 226.04, 240) mm, rotated rx -90 ry -25 rz 121.95 deg; joints [1.28, -47.618, 99.784, 219.529, 108.026, -186.117, -1241.95]
  MoveL 424 to (75.48, 231.77, 250) mm, rotated rx -90 ry -25 rz 126.42 deg; joints [1.626, -47.45, 99.43, 219.71, 108.018, -186.414, -1246.422]
  MoveL 425 to (76.86, 237.05, 260) mm, rotated rx -90 ry -25 rz 130.43 deg; joints [1.97, -47.277, 99.068, 219.888, 108.009, -186.712, -1250.435]
  MoveL 426 to (77.78, 241.77, 270) mm, rotated rx -90 ry -25 rz 133.96 deg; joints [2.312, -47.099, 98.701, 220.065, 108, -187.012, -1253.959]
  MoveL 427 to (78.34, 245.85, 280) mm, rotated rx -90 ry -25 rz 136.96 deg; joints [2.653, -46.916, 98.327, 220.239, 107.991, -187.312, -1256.964]
  MoveL 428 to (78.63, 249.2, 290) mm, rotated rx -90 ry -25 rz 139.42 deg; joints [2.992, -46.728, 97.946, 220.411, 107.981, -187.612, -1259.419]
  MoveL 429 to (58.93, 255.88, 290) mm, rotated rx -90 ry -25 rz 145.69 deg; joints [2.992, -45.858, 98.042, 220.619, 108.716, -186.951, -1265.694]
  Set speed (60.0 mm/s)
  MoveL 430 to (58.94, 253.36, 280) mm, rotated rx -90 ry -25 rz 143.26 deg; joints [2.653, -46.043, 98.422, 220.447, 108.729, -186.651, -1263.258]
  MoveL 431 to (58.8, 250.28, 270) mm, rotated rx -90 ry -25 rz 140.27 deg; joints [2.312, -46.222, 98.796, 220.273, 108.742, -186.351, -1260.274]
  MoveL 432 to (58.44, 246.7, 260) mm, rotated rx -90 ry -25 rz 136.77 deg; joints [1.97, -46.397, 99.163, 220.097, 108.755, -186.052, -1256.77]
  MoveL 433 to (57.77, 242.68, 250) mm, rotated rx -90 ry -25 rz 132.77 deg; joints [1.626, -46.567, 99.524, 219.918, 108.768, -185.755, -1252.774]
  MoveL 434 to (56.69, 238.28, 240) mm, rotated rx -90 ry -25 rz 128.32 deg; joints [1.28, -46.731, 99.878, 219.737, 108.781, -185.458, -1248.316]
  MoveL 435 to (55.14, 233.59, 230) mm, rotated rx -90 ry -25 rz 123.42 deg; joints [0.933, -46.892, 100.226, 219.554, 108.793, -185.162, -1243.424]
  MoveL 436 to (53.04, 228.71, 220) mm, rotated rx -90 ry -25 rz 118.13 deg; joints [0.584, -47.048, 100.567, 219.369, 108.804, -184.868, -1238.126]
  MoveL 437 to (50.33, 223.75, 210) mm, rotated rx -90 ry -25 rz 112.45 deg; joints [0.233, -47.2, 100.902, 219.181, 108.813, -184.576, -1232.453]
  MoveL 438 to (46.98, 218.83, 200) mm, rotated rx -90 ry -25 rz 106.43 deg; joints [-0.119, -47.349, 101.231, 218.99, 108.822, -184.286, -1226.434]
  MoveL 439 to (42.97, 214.08, 190) mm, rotated rx -90 ry -25 rz 100.1 deg; joints [-0.473, -47.495, 101.553, 218.797, 108.828, -183.998, -1220.103]
  MoveL 440 to (38.31, 209.62, 180) mm, rotated rx -90 ry -25 rz 93.49 deg; joints [-0.828, -47.639, 101.869, 218.601, 108.832, -183.713, -1213.494]
  MoveL 441 to (33.03, 205.6, 170) mm, rotated rx -90 ry -25 rz 86.64 deg; joints [-1.185, -47.781, 102.178, 218.402, 108.833, -183.431, -1206.645]
  MoveL 442 to (27.19, 202.13, 160) mm, rotated rx -90 ry -25 rz 79.59 deg; joints [-1.544, -47.922, 102.481, 218.2, 108.831, -183.152, -1199.594]
  MoveL 443 to (20.88, 199.3, 150) mm, rotated rx -90 ry -25 rz 72.38 deg; joints [-1.904, -48.062, 102.777, 217.995, 108.826, -182.877, -1192.384]
  MoveL 444 to (14.2, 197.22, 140) mm, rotated rx -90 ry -25 rz 65.06 deg; joints [-2.265, -48.201, 103.066, 217.788, 108.816, -182.606, -1185.059]
  MoveL 445 to (7.28, 195.93, 130) mm, rotated rx -90 ry -25 rz 57.67 deg; joints [-2.628, -48.34, 103.349, 217.577, 108.802, -182.339, -1177.666]
  MoveL 446 to (0.24, 195.48, 120) mm, rotated rx -90 ry -25 rz 50.25 deg; joints [-2.992, -48.479, 103.625, 217.363, 108.784, -182.076, -1170.252]
  MoveL 447 to (-6.77, 195.87, 110) mm, rotated rx -90 ry -25 rz 42.87 deg; joints [-3.358, -48.619, 103.895, 217.146, 108.762, -181.817, -1162.866]
  MoveL 448 to (-13.63, 197.08, 100) mm, rotated rx -90 ry -25 rz 35.55 deg; joints [-3.725, -48.758, 104.159, 216.926, 108.735, -181.562, -1155.555]
  MoveL 449 to (-20.21, 199.05, 90) mm, rotated rx -90 ry -25 rz 28.37 deg; joints [-4.093, -48.897, 104.415, 216.703, 108.704, -181.311, -1148.366]
  MoveL 450 to (-26.38, 201.72, 80) mm, rotated rx -90 ry -25 rz 21.35 deg; joints [-4.463, -49.036, 104.666, 216.477, 108.669, -181.064, -1141.346]
  MoveL 451 to (-32.08, 204.97, 70) mm, rotated rx -90 ry -25 rz 14.54 deg; joints [-4.834, -49.174, 104.909, 216.248, 108.63, -180.819, -1134.536]
  MoveL 452 to (-37.21, 208.71, 60) mm, rotated rx -90 ry -25 rz 7.98 deg; joints [-5.207, -49.31, 105.147, 216.017, 108.588, -180.578, -1127.979]
  MoveL 453 to (-41.73, 212.8, 50) mm, rotated rx -90 ry -25 rz 1.71 deg; joints [-5.581, -49.445, 105.378, 215.784, 108.543, -180.339, -1121.712]
  MoveL 454 to (-45.64, 217.12, 40) mm, rotated rx -90 ry -25 rz -4.23 deg; joints [-5.956, -49.577, 105.603, 215.548, 108.496, -180.103, -1115.772]
  MoveL 455 to (-48.92, 221.54, 30) mm, rotated rx -90 ry -25 rz -9.81 deg; joints [-6.332, -49.707, 105.821, 215.31, 108.447, -179.868, -1110.192]
  MoveL 456 to (-51.6, 225.93, 20) mm, rotated rx -90 ry -25 rz -15 deg; joints [-6.709, -49.833, 106.033, 215.071, 108.396, -179.635, -1105.005]
  MoveL 457 to (-53.73, 230.19, 10) mm, rotated rx -90 ry -25 rz -19.76 deg; joints [-7.088, -49.956, 106.239, 214.829, 108.344, -179.402, -1100.24]
  MoveL 458 to (-55.37, 234.2, 0) mm, rotated rx -90 ry -25 rz -24.07 deg; joints [-7.468, -50.074, 106.439, 214.586, 108.291, -179.171, -1095.929]
  MoveL 459 to (58.93, 255.88, 290) mm, rotated rx -90 ry -25 rz 145.69 deg; joints [2.992, -45.858, 98.042, 220.619, 108.716, -186.951, -1265.694]
  Set speed (60.0 mm/s)
  MoveL 460 to (37.11, 300.24, 290) mm, rotated rx -90 ry -25 rz -166.45 deg; joints [2.992, -46.004, 98.028, 220.584, 108.594, -187.061, -1313.547]
  MoveL 461 to (-55.37, 234.2, 0) mm, rotated rx -90 ry -25 rz -24.07 deg; joints [-7.468, -50.074, 106.439, 214.586, 108.291, -179.171, -1455.929]
  Set speed (60.0 mm/s)
  MoveL 462 to (-20.49, 199.16, 0) mm, rotated rx -90 ry -25 rz 28.05 deg; joints [-7.468, -49.938, 106.45, 214.613, 108.412, -179.083, -1508.047]
  MoveL 463 to (-55.37, 234.2, 0) mm, rotated rx -90 ry -25 rz -24.07 deg; joints [-7.468, -50.074, 106.439, 214.586, 108.291, -179.171, -1455.929]
  Set speed (60.0 mm/s)
  MoveL 464 to (-53.73, 230.19, 10) mm, rotated rx -90 ry -25 rz -19.76 deg; joints [-7.088, -49.956, 106.239, 214.829, 108.344, -179.402, -1460.24]
  MoveL 465 to (-51.6, 225.93, 20) mm, rotated rx -90 ry -25 rz -15 deg; joints [-6.709, -49.833, 106.033, 215.071, 108.396, -179.635, -1465.005]
  MoveL 466 to (-48.92, 221.54, 30) mm, rotated rx -90 ry -25 rz -9.81 deg; joints [-6.332, -49.707, 105.821, 215.31, 108.447, -179.868, -1470.192]
  MoveL 467 to (-45.64, 217.12, 40) mm, rotated rx -90 ry -25 rz -4.23 deg; joints [-5.956, -49.577, 105.603, 215.548, 108.496, -180.103, -1475.772]
  MoveL 468 to (-41.73, 212.8, 50) mm, rotated rx -90 ry -25 rz 1.71 deg; joints [-5.581, -49.445, 105.378, 215.784, 108.543, -180.339, -1481.712]
  MoveL 469 to (-37.21, 208.71, 60) mm, rotated rx -90 ry -25 rz 7.98 deg; joints [-5.207, -49.31, 105.147, 216.017, 108.588, -180.578, -1487.979]
  MoveL 470 to (-32.08, 204.97, 70) mm, rotated rx -90 ry -25 rz 14.54 deg; joints [-4.834, -49.174, 104.909, 216.248, 108.63, -180.819, -1494.536]
  MoveL 471 to (-26.38, 201.72, 80) mm, rotated rx -90 ry -25 rz 21.35 deg; joints [-4.463, -49.036, 104.666, 216.477, 108.669, -181.064, -1501.346]
  MoveL 472 to (-20.21, 199.05, 90) mm, rotated rx -90 ry -25 rz 28.37 deg; joints [-4.093, -48.897, 104.415, 216.703, 108.704, -181.311, -1508.366]
  MoveL 473 to (-13.63, 197.08, 100) mm, rotated rx -90 ry -25 rz 35.55 deg; joints [-3.725, -48.758, 104.159, 216.926, 108.735, -181.562, -1515.555]
  MoveL 474 to (-6.77, 195.87, 110) mm, rotated rx -90 ry -25 rz 42.87 deg; joints [-3.358, -48.619, 103.895, 217.146, 108.762, -181.817, -1522.866]
  MoveL 475 to (0.24, 195.48, 120) mm, rotated rx -90 ry -25 rz 50.25 deg; joints [-2.992, -48.479, 103.625, 217.363, 108.784, -182.076, -1530.252]
  MoveL 476 to (7.28, 195.93, 130) mm, rotated rx -90 ry -25 rz 57.67 deg; joints [-2.628, -48.34, 103.349, 217.577, 108.802, -182.339, -1537.666]
  MoveL 477 to (14.2, 197.22, 140) mm, rotated rx -90 ry -25 rz 65.06 deg; joints [-2.265, -48.201, 103.066, 217.788, 108.816, -182.606, -1545.059]
  MoveL 478 to (20.88, 199.3, 150) mm, rotated rx -90 ry -25 rz 72.38 deg; joints [-1.904, -48.062, 102.777, 217.995, 108.826, -182.877, -1552.384]
  MoveL 479 to (27.19, 202.13, 160) mm, rotated rx -90 ry -25 rz 79.59 deg; joints [-1.544, -47.922, 102.481, 218.2, 108.831, -183.152, -1559.594]
  MoveL 480 to (33.03, 205.6, 170) mm, rotated rx -90 ry -25 rz 86.64 deg; joints [-1.185, -47.781, 102.178, 218.402, 108.833, -183.431, -1566.645]
  MoveL 481 to (38.31, 209.62, 180) mm, rotated rx -90 ry -25 rz 93.49 deg; joints [-0.828, -47.639, 101.869, 218.601, 108.832, -183.713, -1573.494]
  MoveL 482 to (42.97, 214.08, 190) mm, rotated rx -90 ry -25 rz 100.1 deg; joints [-0.473, -47.495, 101.553, 218.797, 108.828, -183.998, -1580.103]
  MoveL 483 to (46.98, 218.83, 200) mm, rotated rx -90 ry -25 rz 106.43 deg; joints [-0.119, -47.349, 101.231, 218.99, 108.822, -184.286, -1586.434]
  MoveL 484 to (50.33, 223.75, 210) mm, rotated rx -90 ry -25 rz 112.45 deg; joints [0.233, -47.2, 100.902, 219.181, 108.813, -184.576, -1592.453]
  MoveL 485 to (53.04, 228.71, 220) mm, rotated rx -90 ry -25 rz 118.13 deg; joints [0.584, -47.048, 100.567, 219.369, 108.804, -184.868, -1598.126]
  MoveL 486 to (55.14, 233.59, 230) mm, rotated rx -90 ry -25 rz 123.42 deg; joints [0.933, -46.892, 100.226, 219.554, 108.793, -185.162, -1603.424]
  MoveL 487 to (56.69, 238.28, 240) mm, rotated rx -90 ry -25 rz 128.32 deg; joints [1.28, -46.731, 99.878, 219.737, 108.781, -185.458, -1608.316]
  MoveL 488 to (57.77, 242.68, 250) mm, rotated rx -90 ry -25 rz 132.77 deg; joints [1.626, -46.567, 99.524, 219.918, 108.768, -185.755, -1612.774]
  MoveL 489 to (58.44, 246.7, 260) mm, rotated rx -90 ry -25 rz 136.77 deg; joints [1.97, -46.397, 99.163, 220.097, 108.755, -186.052, -1616.77]
  MoveL 490 to (58.8, 250.28, 270) mm, rotated rx -90 ry -25 rz 140.27 deg; joints [2.312, -46.222, 98.796, 220.273, 108.742, -186.351, -1620.274]
  MoveL 491 to (58.94, 253.36, 280) mm, rotated rx -90 ry -25 rz 143.26 deg; joints [2.653, -46.043, 98.422, 220.447, 108.729, -186.651, -1623.258]
  MoveL 492 to (58.93, 255.88, 290) mm, rotated rx -90 ry -25 rz 145.69 deg; joints [2.992, -45.858, 98.042, 220.619, 108.716, -186.951, -1625.694]
  MoveL 493 to (37.11, 300.24, 290) mm, rotated rx -96.9 ry -17.88 rz 75.79 deg; joints [-1.762, -22.307, 19.15, 321.67, 56.455, -329.47, -1646.629]
  Set speed (60.0 mm/s)
  MoveL 494 to (39.03, 298.61, 280) mm, rotated rx -97.08 ry -15.54 rz 79.68 deg; joints [-1.817, -34.316, 42.197, 311.116, 41.994, -315.035, -1643.609]
  MoveL 495 to (41.29, 296.51, 270) mm, rotated rx -98.79 ry -14.56 rz 73.06 deg; joints [-2.194, -31.58, 37.029, 317.372, 44.628, -323.492, -1640.035]
  MoveL 496 to (43.78, 293.91, 260) mm, rotated rx -100.6 ry -13.96 rz 65.48 deg; joints [-2.524, -27.364, 29.096, 323.507, 49.428, -332.28, -1635.959]
  MoveL 497 to (44.93, 293.38, 249.12) mm, rotated rx -102.48 ry -13.76 rz 57.03 deg; joints [-2.804, -17.515, 10.028, 330.069, 60.063, -343.189, -1631.425]
  MoveL 498 to (49.06, 287.12, 240) mm, rotated rx -102.2 ry -11.88 rz 56.85 deg; joints [-3.056, -30.478, 35.086, 323.792, 44.843, -332.966, -1626.478]
  MoveL 499 to (51.62, 282.9, 230) mm, rotated rx -75.3 ry -12.71 rz 137.52 deg; joints [-3.935, -50.762, 109.257, 204.608, 107.196, -170.197, -1621.161]
  MoveL 500 to (53.98, 278.14, 220) mm, rotated rx -73.63 ry -13.16 rz 135.62 deg; joints [-4.597, -49.036, 109.478, 204.655, 112.497, -166.43, -1615.515]
  MoveL 501 to (56, 272.86, 210) mm, rotated rx -72.12 ry -13.76 rz 133.16 deg; joints [-5.21, -47.279, 109.363, 205.11, 117.258, -162.823, -1609.582]
  MoveL 502 to (57.57, 267.12, 200) mm, rotated rx -73 ry -11.66 rz 121.38 deg; joints [-5.837, -50.269, 110.344, 202.253, 109.766, -166.343, -1603.4]
  MoveL 503 to (58.59, 260.98, 190) mm, rotated rx -71.71 ry -12.29 rz 118.09 deg; joints [-6.387, -48.731, 110.34, 202.647, 114.135, -163.303, -1597.009]
  MoveL 504 to (58.95, 254.55, 180) mm, rotated rx -70.55 ry -13.02 rz 114.47 deg; joints [-6.895, -47.173, 110.109, 203.335, 118.142, -160.337, -1590.447]
  MoveL 505 to (58.59, 247.92, 170) mm, rotated rx -71.88 ry -10.84 rz 101.84 deg; joints [-7.456, -50.401, 111.102, 200.323, 110.121, -164.461, -1583.752]
  MoveL 506 to (57.45, 241.22, 160) mm, rotated rx -70.86 ry -11.6 rz 97.82 deg; joints [-7.918, -48.992, 111.026, 200.911, 114.028, -161.903, -1576.959]
  MoveL 507 to (55.51, 234.59, 150) mm, rotated rx -69.95 ry -12.44 rz 93.68 deg; joints [-8.342, -47.538, 110.762, 201.759, 117.727, -159.341, -1570.107]
  MoveL 508 to (52.77, 228.15, 140) mm, rotated rx -71.59 ry -10.32 rz 80.79 deg; joints [-8.837, -50.822, 111.649, 198.83, 109.469, -163.735, -1563.231]
  MoveL 509 to (49.26, 222.05, 130) mm, rotated rx -70.76 ry -11.22 rz 76.66 deg; joints [-9.222, -49.431, 111.542, 199.623, 113.329, -161.424, -1556.367]
  MoveL 510 to (45.04, 216.4, 120) mm, rotated rx -70.03 ry -12.23 rz 72.63 deg; joints [-9.569, -47.95, 111.245, 200.697, 117.11, -159.03, -1549.55]
  MoveL 511 to (40.19, 211.31, 110) mm, rotated rx -71.83 ry -10.32 rz 60.03 deg; joints [-9.99, -51.146, 112.007, 198.026, 108.991, -163.457, -1542.816]
  MoveL 512 to (34.83, 206.87, 100) mm, rotated rx -71.13 ry -11.44 rz 56.41 deg; joints [-10.295, -49.635, 111.85, 199.132, 113.184, -161.164, -1536.2]
  MoveL 513 to (29.06, 203.14, 90) mm, rotated rx -70.54 ry -12.69 rz 53.09 deg; joints [-10.556, -47.975, 111.465, 200.587, 117.401, -158.693, -1529.736]
  MoveL 514 to (23.03, 200.17, 80) mm, rotated rx -72.37 ry -11.13 rz 41.37 deg; joints [-10.892, -50.973, 112.184, 198.264, 109.884, -163.026, -1523.458]
  MoveL 515 to (16.86, 197.94, 70) mm, rotated rx -71.8 ry -12.55 rz 38.86 deg; joints [-11.1, -49.174, 111.89, 199.878, 114.745, -160.508, -1517.4]
  MoveL 516 to (10.69, 196.46, 60) mm, rotated rx -73.66 ry -11.39 rz 28.02 deg; joints [-11.348, -51.869, 112.326, 198.148, 107.646, -164.538, -1511.595]
  MoveL 517 to (4.64, 195.67, 50) mm, rotated rx -73.16 ry -13.02 rz 26.6 deg; joints [-11.489, -49.859, 112.079, 200.024, 113.289, -161.87, -1506.075]
  MoveL 518 to (-1.18, 195.49, 40) mm, rotated rx -74.98 ry -12.29 rz 16.89 deg; joints [-11.645, -52.231, 112.35, 198.85, 106.89, -165.63, -1500.872]
  MoveL 519 to (-6.67, 195.86, 30) mm, rotated rx -74.62 ry -14.16 rz 16.83 deg; joints [-11.702, -49.919, 112.059, 201.112, 113.427, -162.696, -1496.017]
  MoveL 520 to (-11.76, 196.67, 20) mm, rotated rx -76.4 ry -13.89 rz 8.51 deg; joints [-11.758, -51.951, 112.266, 200.461, 107.995, -166.208, -1491.54]
  MoveL 521 to (-16.38, 197.8, 10) mm, rotated rx -78.17 ry -13.98 rz 0.96 deg; joints [-11.742, -53.642, 112.118, 200.427, 102.896, -169.457, -1487.469]
  MoveL 522 to (-20.49, 199.16, 0) mm, rotated rx -78.17 ry -13.98 rz 0.96 deg; joints [-12.168, -53.619, 111.889, 200.096, 102.626, -169.315, -1487.469]
  MoveL 523 to (37.11, 300.24, 290) mm, rotated rx -90 ry -25 rz -166.45 deg; joints [2.992, -46.004, 98.028, 220.584, 108.594, -187.061, -1313.547]
  Set speed (60.0 mm/s)
  MoveL 524 to (43.85, 319.91, 290) mm, rotated rx -90 ry -25 rz -162.09 deg; joints [2.992, -46.901, 97.924, 220.37, 107.832, -187.745, -1317.907]
  MoveL 525 to (-20.49, 199.16, 0) mm, rotated rx -90 ry -25 rz 28.05 deg; joints [-7.468, -49.938, 106.45, 214.613, 108.412, -179.083, -1148.047]
  Set speed (60.0 mm/s)
  MoveL 526 to (-20.57, 178.36, 0) mm, rotated rx -90 ry -25 rz 33.98 deg; joints [-7.468, -50.9, 106.359, 214.42, 107.545, -179.71, -1153.977]
  MoveL 527 to (-20.49, 199.16, 0) mm, rotated rx -90 ry -25 rz 28.05 deg; joints [-7.468, -49.938, 106.45, 214.613, 108.412, -179.083, -1148.047]
  Set speed (60.0 mm/s)
  MoveL 528 to (-16.38, 197.8, 10) mm, rotated rx -90 ry -25 rz 32.58 deg; joints [-7.088, -49.83, 106.249, 214.855, 108.455, -179.321, -1152.579]
  MoveL 529 to (-11.76, 196.67, 20) mm, rotated rx -90 ry -25 rz 37.57 deg; joints [-6.709, -49.719, 106.042, 215.094, 108.496, -179.56, -1157.568]
  MoveL 530 to (-6.67, 195.86, 30) mm, rotated rx -90 ry -25 rz 42.97 deg; joints [-6.332, -49.607, 105.829, 215.331, 108.535, -179.802, -1162.975]
  MoveL 531 to (-1.18, 195.49, 40) mm, rotated rx -90 ry -25 rz 48.76 deg; joints [-5.956, -49.493, 105.609, 215.566, 108.57, -180.047, -1168.76]
  MoveL 532 to (4.64, 195.67, 50) mm, rotated rx -90 ry -25 rz 54.88 deg; joints [-5.581, -49.378, 105.383, 215.798, 108.602, -180.295, -1174.88]
  MoveL 533 to (10.69, 196.46, 60) mm, rotated rx -90 ry -25 rz 61.29 deg; joints [-5.207, -49.263, 105.151, 216.028, 108.63, -180.546, -1181.291]
  MoveL 534 to (16.86, 197.94, 70) mm, rotated rx -90 ry -25 rz 67.95 deg; joints [-4.834, -49.146, 104.912, 216.254, 108.654, -180.801, -1187.947]
  MoveL 535 to (23.03, 200.17, 80) mm, rotated rx -90 ry -25 rz 74.8 deg; joints [-4.463, -49.03, 104.666, 216.478, 108.674, -181.059, -1194.802]
  MoveL 536 to (29.06, 203.14, 90) mm, rotated rx -90 ry -25 rz 81.81 deg; joints [-4.093, -48.913, 104.414, 216.699, 108.69, -181.322, -1201.809]
  MoveL 537 to (34.83, 206.87, 100) mm, rotated rx -90 ry -25 rz 88.92 deg; joints [-3.725, -48.796, 104.156, 216.917, 108.702, -181.588, -1208.92]
  MoveL 538 to (40.19, 211.31, 110) mm, rotated rx -90 ry -25 rz 96.09 deg; joints [-3.358, -48.678, 103.891, 217.133, 108.711, -181.858, -1216.089]
  MoveL 539 to (45.04, 216.4, 120) mm, rotated rx -90 ry -25 rz 103.27 deg; joints [-2.992, -48.56, 103.619, 217.345, 108.716, -182.131, -1223.271]
  MoveL 540 to (49.26, 222.05, 130) mm, rotated rx -90 ry -25 rz 110.42 deg; joints [-2.628, -48.44, 103.341, 217.555, 108.717, -182.408, -1230.424]
  MoveL 541 to (52.77, 228.15, 140) mm, rotated rx -90 ry -25 rz 117.51 deg; joints [-2.265, -48.318, 103.057, 217.761, 108.716, -182.687, -1237.506]
  MoveL 542 to (55.51, 234.59, 150) mm, rotated rx -90 ry -25 rz 124.48 deg; joints [-1.904, -48.193, 102.766, 217.966, 108.713, -182.97, -1244.481]
  MoveL 543 to (57.45, 241.22, 160) mm, rotated rx -90 ry -25 rz 131.31 deg; joints [-1.544, -48.066, 102.469, 218.167, 108.708, -183.254, -1251.311]
  MoveL 544 to (58.59, 247.92, 170) mm, rotated rx -90 ry -25 rz 137.96 deg; joints [-1.185, -47.936, 102.165, 218.366, 108.701, -183.541, -1257.965]
  MoveL 545 to (58.95, 254.55, 180) mm, rotated rx -90 ry -25 rz 144.41 deg; joints [-0.828, -47.802, 101.855, 218.563, 108.694, -183.829, -1264.41]
  MoveL 546 to (58.59, 260.98, 190) mm, rotated rx -90 ry -25 rz 150.62 deg; joints [-0.473, -47.664, 101.539, 218.758, 108.685, -184.119, -1270.617]
  MoveL 547 to (57.57, 267.12, 200) mm, rotated rx -90 ry -25 rz 156.56 deg; joints [-0.119, -47.521, 101.216, 218.95, 108.677, -184.409, -1276.558]
  MoveL 548 to (56, 272.86, 210) mm, rotated rx -90 ry -25 rz 162.2 deg; joints [0.233, -47.373, 100.887, 219.14, 108.668, -184.701, -1282.205]
  MoveL 549 to (53.98, 278.14, 220) mm, rotated rx -90 ry -25 rz 167.53 deg; joints [0.584, -47.22, 100.552, 219.328, 108.659, -184.994, -1287.531]
  MoveL 550 to (51.62, 282.9, 230) mm, rotated rx -90 ry -25 rz 172.51 deg; joints [0.933, -47.062, 100.211, 219.514, 108.65, -185.287, -1292.509]
  MoveL 551 to (49.06, 287.12, 240) mm, rotated rx -90 ry -25 rz 177.11 deg; joints [1.28, -46.898, 99.863, 219.698, 108.641, -185.581, -1297.114]
  MoveL 552 to (46.4, 290.79, 250) mm, rotated rx -90 ry -25 rz -178.68 deg; joints [1.626, -46.729, 99.509, 219.879, 108.632, -185.875, -1301.316]
  MoveL 553 to (43.78, 293.91, 260) mm, rotated rx -90 ry -25 rz -174.91 deg; joints [1.97, -46.556, 99.148, 220.059, 108.623, -186.17, -1305.09]
  MoveL 554 to (41.29, 296.51, 270) mm, rotated rx -90 ry -25 rz -171.59 deg; joints [2.312, -46.377, 98.781, 220.236, 108.614, -186.466, -1308.405]
  MoveL 555 to (39.03, 298.61, 280) mm, rotated rx -90 ry -25 rz -168.77 deg; joints [2.653, -46.193, 98.408, 220.411, 108.604, -186.763, -1311.234]
  MoveL 556 to (37.11, 300.24, 290) mm, rotated rx -90 ry -25 rz -166.45 deg; joints [2.992, -46.004, 98.028, 220.584, 108.594, -187.061, -1313.547]
  MoveL 557 to (43.85, 319.91, 290) mm, rotated rx -90 ry -25 rz -162.09 deg; joints [2.992, -46.901, 97.924, 220.37, 107.832, -187.745, -1317.907]
  Set speed (60.0 mm/s)
  MoveL 558 to (46.6, 317.98, 280) mm, rotated rx -90 ry -25 rz -164.43 deg; joints [2.653, -47.093, 98.303, 220.197, 107.838, -187.447, -1315.567]
  MoveL 559 to (49.86, 315.46, 270) mm, rotated rx -90 ry -25 rz -167.29 deg; joints [2.312, -47.281, 98.677, 220.022, 107.842, -187.151, -1312.706]
  MoveL 560 to (53.49, 312.31, 260) mm, rotated rx -90 ry -25 rz -170.65 deg; joints [1.97, -47.464, 99.044, 219.845, 107.847, -186.855, -1309.355]
  MoveL 561 to (57.36, 308.47, 250) mm, rotated rx -90 ry -25 rz -174.45 deg; joints [1.626, -47.641, 99.405, 219.665, 107.851, -186.559, -1305.545]
  MoveL 562 to (61.34, 303.9, 240) mm, rotated rx -90 ry -25 rz -178.69 deg; joints [1.28, -47.814, 99.759, 219.484, 107.855, -186.265, -1301.306]
  MoveL 563 to (65.27, 298.59, 230) mm, rotated rx -90 ry -25 rz 176.67 deg; joints [0.933, -47.981, 100.107, 219.3, 107.859, -185.97, -1296.668]
  MoveL 564 to (68.98, 292.54, 220) mm, rotated rx -90 ry -25 rz 171.66 deg; joints [0.584, -48.143, 100.449, 219.114, 107.864, -185.677, -1291.66]
  MoveL 565 to (72.31, 285.76, 210) mm, rotated rx -90 ry -25 rz 166.31 deg; joints [0.233, -48.3, 100.785, 218.926, 107.868, -185.384, -1286.311]
  MoveL 566 to (75.1, 278.3, 200) mm, rotated rx -90 ry -25 rz 160.65 deg; joints [-0.119, -48.452, 101.115, 218.736, 107.872, -185.092, -1280.65]
  MoveL 567 to (77.2, 270.26, 190) mm, rotated rx -90 ry -25 rz 154.71 deg; joints [-0.473, -48.599, 101.438, 218.544, 107.877, -184.8, -1274.706]
  MoveL 568 to (78.47, 261.74, 180) mm, rotated rx -90 ry -25 rz 148.51 deg; joints [-0.828, -48.74, 101.755, 218.35, 107.881, -184.509, -1268.508]
  MoveL 569 to (78.79, 252.87, 170) mm, rotated rx -90 ry -25 rz 142.09 deg; joints [-1.185, -48.878, 102.066, 218.153, 107.884, -184.22, -1262.086]
  MoveL 570 to (78.09, 243.82, 160) mm, rotated rx -90 ry -25 rz 135.47 deg; joints [-1.544, -49.011, 102.37, 217.955, 107.887, -183.932, -1255.472]
  MoveL 571 to (76.31, 234.75, 150) mm, rotated rx -90 ry -25 rz 128.7 deg; joints [-1.904, -49.141, 102.668, 217.753, 107.888, -183.645, -1248.696]
  MoveL 572 to (73.44, 225.85, 140) mm, rotated rx -90 ry -25 rz 121.79 deg; joints [-2.265, -49.268, 102.96, 217.55, 107.888, -183.361, -1241.794]
  MoveL 573 to (69.5, 217.29, 130) mm, rotated rx -90 ry -25 rz 114.8 deg; joints [-2.628, -49.392, 103.245, 217.344, 107.885, -183.079, -1234.8]
  MoveL 574 to (64.57, 209.26, 120) mm, rotated rx -90 ry -25 rz 107.75 deg; joints [-2.992, -49.514, 103.524, 217.135, 107.88, -182.8, -1227.751]
  MoveL 575 to (58.74, 201.9, 110) mm, rotated rx -90 ry -25 rz 100.69 deg; joints [-3.358, -49.634, 103.796, 216.924, 107.872, -182.524, -1220.687]
  MoveL 576 to (52.14, 195.34, 100) mm, rotated rx -90 ry -25 rz 93.65 deg; joints [-3.725, -49.753, 104.062, 216.709, 107.861, -182.251, -1213.646]
  MoveL 577 to (44.91, 189.68, 90) mm, rotated rx -90 ry -25 rz 86.67 deg; joints [-4.093, -49.872, 104.321, 216.492, 107.846, -181.982, -1206.671]
  MoveL 578 to (37.24, 184.98, 80) mm, rotated rx -90 ry -25 rz 79.81 deg; joints [-4.463, -49.989, 104.574, 216.273, 107.827, -181.716, -1199.806]
  MoveL 579 to (29.3, 181.28, 70) mm, rotated rx -90 ry -25 rz 73.09 deg; joints [-4.834, -50.106, 104.82, 216.05, 107.805, -181.454, -1193.092]
  MoveL 580 to (21.27, 178.55, 60) mm, rotated rx -90 ry -25 rz 66.58 deg; joints [-5.207, -50.223, 105.059, 215.825, 107.778, -181.196, -1186.575]
  MoveL 581 to (13.31, 176.76, 50) mm, rotated rx -90 ry -25 rz 60.3 deg; joints [-5.581, -50.339, 105.292, 215.597, 107.748, -180.941, -1180.298]
  MoveL 582 to (5.58, 175.83, 40) mm, rotated rx -90 ry -25 rz 54.3 deg; joints [-5.956, -50.454, 105.518, 215.366, 107.714, -180.689, -1174.303]
  MoveL 583 to (-1.77, 175.65, 30) mm, rotated rx -90 ry -25 rz 48.63 deg; joints [-6.332, -50.568, 105.738, 215.133, 107.676, -180.44, -1168.634]
  MoveL 584 to (-8.64, 176.1, 20) mm, rotated rx -90 ry -25 rz 43.33 deg; joints [-6.709, -50.68, 105.952, 214.897, 107.635, -180.195, -1163.33]
  MoveL 585 to (-14.93, 177.06, 10) mm, rotated rx -90 ry -25 rz 38.43 deg; joints [-7.088, -50.791, 106.159, 214.66, 107.591, -179.951, -1158.431]
  MoveL 586 to (-20.57, 178.36, 0) mm, rotated rx -90 ry -25 rz 33.98 deg; joints [-7.468, -50.9, 106.359, 214.42, 107.545, -179.71, -1153.977]
  MoveL 587 to (43.85, 319.91, 290) mm, rotated rx -90 ry -25 rz -162.09 deg; joints [2.992, -46.901, 97.924, 220.37, 107.832, -187.745, -1317.907]
  Set speed (60.0 mm/s)
  MoveL 588 to (28.22, 306.19, 290) mm, rotated rx -90 ry -25 rz -156.66 deg; joints [2.992, -46.023, 98.026, 220.579, 108.578, -187.075, -1323.337]
  MoveL 589 to (-20.57, 178.36, 0) mm, rotated rx -90 ry -25 rz 33.98 deg; joints [-7.468, -50.9, 106.359, 214.42, 107.545, -179.71, -1153.977]
  Set speed (60.0 mm/s)
  MoveL 590 to (-10.16, 196.36, 0) mm, rotated rx -90 ry -25 rz 39.27 deg; joints [-7.468, -49.927, 106.451, 214.616, 108.422, -179.076, -1159.273]
  MoveL 591 to (-20.57, 178.36, 0) mm, rotated rx -90 ry -25 rz 33.98 deg; joints [-7.468, -50.9, 106.359, 214.42, 107.545, -179.71, -1153.977]
  Set speed (60.0 mm/s)
  MoveL 592 to (-14.93, 177.06, 10) mm, rotated rx -90 ry -25 rz 38.43 deg; joints [-7.088, -50.791, 106.159, 214.66, 107.591, -179.951, -1158.431]
  MoveL 593 to (-8.64, 176.1, 20) mm, rotated rx -90 ry -25 rz 43.33 deg; joints [-6.709, -50.68, 105.952, 214.897, 107.635, -180.195, -1163.33]
  MoveL 594 to (-1.77, 175.65, 30) mm, rotated rx -90 ry -25 rz 48.63 deg; joints [-6.332, -50.568, 105.738, 215.133, 107.676, -180.44, -1168.634]
  MoveL 595 to (5.58, 175.83, 40) mm, rotated rx -90 ry -25 rz 54.3 deg; joints [-5.956, -50.454, 105.518, 215.366, 107.714, -180.689, -1174.303]
  MoveL 596 to (13.31, 176.76, 50) mm, rotated rx -90 ry -25 rz 60.3 deg; joints [-5.581, -50.339, 105.292, 215.597, 107.748, -180.941, -1180.298]
  MoveL 597 to (21.27, 178.55, 60) mm, rotated rx -90 ry -25 rz 66.58 deg; joints [-5.207, -50.223, 105.059, 215.825, 107.778, -181.196, -1186.575]
  MoveL 598 to (29.3, 181.28, 70) mm, rotated rx -90 ry -25 rz 73.09 deg; joints [-4.834, -50.106, 104.82, 216.05, 107.805, -181.454, -1193.092]
  MoveL 599 to (37.24, 184.98, 80) mm, rotated rx -90 ry -25 rz 79.81 deg; joints [-4.463, -49.989, 104.574, 216.273, 107.827, -181.716, -1199.806]
  MoveL 600 to (44.91, 189.68, 90) mm, rotated rx -90 ry -25 rz 86.67 deg; joints [-4.093, -49.872, 104.321, 216.492, 107.846, -181.982, -1206.671]
  MoveL 601 to (52.14, 195.34, 100) mm, rotated rx -90 ry -25 rz 93.65 deg; joints [-3.725, -49.753, 104.062, 216.709, 107.861, -182.251, -1213.646]
  MoveL 602 to (58.74, 201.9, 110) mm, rotated rx -90 ry -25 rz 100.69 deg; joints [-3.358, -49.634, 103.796, 216.924, 107.872, -182.524, -1220.687]
  MoveL 603 to (64.57, 209.26, 120) mm, rotated rx -90 ry -25 rz 107.75 deg; joints [-2.992, -49.514, 103.524, 217.135, 107.88, -182.8, -1227.751]
  MoveL 604 to (69.5, 217.29, 130) mm, rotated rx -90 ry -25 rz 114.8 deg; joints [-2.628, -49.392, 103.245, 217.344, 107.885, -183.079, -1234.8]
  MoveL 605 to (73.44, 225.85, 140) mm, rotated rx -90 ry -25 rz 121.79 deg; joints [-2.265, -49.268, 102.96, 217.55, 107.888, -183.361, -1241.794]
  MoveL 606 to (76.31, 234.75, 150) mm, rotated rx -90 ry -25 rz 128.7 deg; joints [-1.904, -49.141, 102.668, 217.753, 107.888, -183.645, -1248.696]
  MoveL 607 to (78.09, 243.82, 160) mm, rotated rx -90 ry -25 rz 135.47 deg; joints [-1.544, -49.011, 102.37, 217.955, 107.887, -183.932, -1255.472]
  MoveL 608 to (78.79, 252.87, 170) mm, rotated rx -90 ry -25 rz 142.09 deg; joints [-1.185, -48.878, 102.066, 218.153, 107.884, -184.22, -1262.086]
  MoveL 609 to (78.47, 261.74, 180) mm, rotated rx -90 ry -25 rz 148.51 deg; joints [-0.828, -48.74, 101.755, 218.35, 107.881, -184.509, -1268.508]
  MoveL 610 to (77.2, 270.26, 190) mm, rotated rx -90 ry -25 rz 154.71 deg; joints [-0.473, -48.599, 101.438, 218.544, 107.877, -184.8, -1274.706]
  MoveL 611 to (75.1, 278.3, 200) mm, rotated rx -90 ry -25 rz 160.65 deg; joints [-0.119, -48.452, 101.115, 218.736, 107.872, -185.092, -1280.65]
  MoveL 612 to (72.31, 285.76, 210) mm, rotated rx -90 ry -25 rz 166.31 deg; joints [0.233, -48.3, 100.785, 218.926, 107.868, -185.384, -1286.311]
  MoveL 613 to (68.98, 292.54, 220) mm, rotated rx -90 ry -25 rz 171.66 deg; joints [0.584, -48.143, 100.449, 219.114, 107.864, -185.677, -1291.66]
  MoveL 614 to (65.27, 298.59, 230) mm, rotated rx -90 ry -25 rz 176.67 deg; joints [0.933, -47.981, 100.107, 219.3, 107.859, -185.97, -1296.668]
  MoveL 615 to (61.34, 303.9, 240) mm, rotated rx -90 ry -25 rz -178.69 deg; joints [1.28, -47.814, 99.759, 219.484, 107.855, -186.265, -1301.306]
  MoveL 616 to (57.36, 308.47, 250) mm, rotated rx -90 ry -25 rz -174.45 deg; joints [1.626, -47.641, 99.405, 219.665, 107.851, -186.559, -1305.545]
  MoveL 617 to (53.49, 312.31, 260) mm, rotated rx -90 ry -25 rz -170.65 deg; joints [1.97, -47.464, 99.044, 219.845, 107.847, -186.855, -1309.355]
  MoveL 618 to (49.86, 315.46, 270) mm, rotated rx -90 ry -25 rz -167.29 deg; joints [2.312, -47.281, 98.677, 220.022, 107.842, -187.151, -1312.706]
  MoveL 619 to (46.6, 317.98, 280) mm, rotated rx -90 ry -25 rz -164.43 deg; joints [2.653, -47.093, 98.303, 220.197, 107.838, -187.447, -1315.567]
  MoveL 620 to (43.85, 319.91, 290) mm, rotated rx -90 ry -25 rz -162.09 deg; joints [2.992, -46.901, 97.924, 220.37, 107.832, -187.745, -1317.907]
  MoveL 621 to (28.22, 306.19, 290) mm, rotated rx -90 ry -25 rz -156.66 deg; joints [2.992, -46.023, 98.026, 220.579, 108.578, -187.075, -1323.337]
  Set speed (60.0 mm/s)
  MoveL 622 to (30.4, 304.94, 280) mm, rotated rx -90 ry -25 rz -158.96 deg; joints [2.653, -46.213, 98.406, 220.406, 108.587, -186.778, -1321.04]
  MoveL 623 to (33, 303.28, 270) mm, rotated rx -90 ry -25 rz -161.77 deg; joints [2.312, -46.398, 98.779, 220.231, 108.595, -186.483, -1318.23]
  MoveL 624 to (35.92, 301.18, 260) mm, rotated rx -90 ry -25 rz -165.06 deg; joints [1.97, -46.579, 99.146, 220.053, 108.603, -186.188, -1314.94]
  MoveL 625 to (39.07, 298.58, 250) mm, rotated rx -90 ry -25 rz -168.8 deg; joints [1.626, -46.755, 99.506, 219.873, 108.61, -185.894, -1311.197]
  MoveL 626 to (42.34, 295.45, 240) mm, rotated rx -90 ry -25 rz -172.97 deg; joints [1.28, -46.926, 99.86, 219.691, 108.618, -185.601, -1307.031]
  MoveL 627 to (45.62, 291.76, 230) mm, rotated rx -90 ry -25 rz -177.53 deg; joints [0.933, -47.091, 100.208, 219.507, 108.625, -185.308, -1302.471]
  MoveL 628 to (48.8, 287.5, 220) mm, rotated rx -90 ry -25 rz 177.54 deg; joints [0.584, -47.251, 100.549, 219.321, 108.632, -185.016, -1297.543]
  MoveL 629 to (51.74, 282.68, 210) mm, rotated rx -90 ry -25 rz 172.28 deg; joints [0.233, -47.406, 100.884, 219.133, 108.64, -184.725, -1292.275]
  MoveL 630 to (54.33, 277.32, 200) mm, rotated rx -90 ry -25 rz 166.69 deg; joints [-0.119, -47.555, 101.213, 218.942, 108.647, -184.435, -1286.694]
  MoveL 631 to (56.44, 271.47, 190) mm, rotated rx -90 ry -25 rz 160.83 deg; joints [-0.473, -47.7, 101.535, 218.75, 108.655, -184.145, -1280.826]
  MoveL 632 to (57.96, 265.2, 180) mm, rotated rx -90 ry -25 rz 154.7 deg; joints [-0.828, -47.839, 101.852, 218.555, 108.662, -183.856, -1274.699]
  MoveL 633 to (58.8, 258.62, 170) mm, rotated rx -90 ry -25 rz 148.34 deg; joints [-1.185, -47.974, 102.162, 218.358, 108.669, -183.568, -1268.339]
  MoveL 634 to (58.89, 251.83, 160) mm, rotated rx -90 ry -25 rz 141.78 deg; joints [-1.544, -48.104, 102.465, 218.159, 108.676, -183.281, -1261.776]
  MoveL 635 to (58.18, 244.95, 150) mm, rotated rx -90 ry -25 rz 135.04 deg; joints [-1.904, -48.231, 102.763, 217.957, 108.681, -182.996, -1255.039]
  MoveL 636 to (56.65, 238.12, 140) mm, rotated rx -90 ry -25 rz 128.16 deg; joints [-2.265, -48.354, 103.054, 217.753, 108.685, -182.713, -1248.16]
  MoveL 637 to (54.3, 231.49, 130) mm, rotated rx -90 ry -25 rz 121.17 deg; joints [-2.628, -48.474, 103.338, 217.547, 108.687, -182.432, -1241.173]
  MoveL 638 to (51.17, 225.17, 120) mm, rotated rx -90 ry -25 rz 114.11 deg; joints [-2.992, -48.592, 103.616, 217.338, 108.687, -182.154, -1234.112]
  MoveL 639 to (47.33, 219.29, 110) mm, rotated rx -90 ry -25 rz 107.02 deg; joints [-3.358, -48.708, 103.888, 217.126, 108.685, -181.879, -1227.017]
  MoveL 640 to (42.85, 213.95, 100) mm, rotated rx -90 ry -25 rz 99.93 deg; joints [-3.725, -48.823, 104.153, 216.911, 108.679, -181.606, -1219.928]
  MoveL 641 to (37.86, 209.24, 90) mm, rotated rx -90 ry -25 rz 92.89 deg; joints [-4.093, -48.937, 104.412, 216.694, 108.67, -181.338, -1212.888]
  MoveL 642 to (32.46, 205.23, 80) mm, rotated rx -90 ry -25 rz 85.94 deg; joints [-4.463, -49.05, 104.664, 216.474, 108.657, -181.073, -1205.942]
  MoveL 643 to (26.8, 201.92, 70) mm, rotated rx -90 ry -25 rz 79.14 deg; joints [-4.834, -49.162, 104.91, 216.251, 108.64, -180.811, -1199.135]
  MoveL 644 to (21, 199.35, 60) mm, rotated rx -90 ry -25 rz 72.51 deg; joints [-5.207, -49.274, 105.15, 216.025, 108.62, -180.554, -1192.515]
  MoveL 645 to (15.19, 197.47, 50) mm, rotated rx -90 ry -25 rz 66.13 deg; joints [-5.581, -49.385, 105.383, 215.797, 108.596, -180.3, -1186.127]
  MoveL 646 to (9.5, 196.25, 40) mm, rotated rx -90 ry -25 rz 60.02 deg; joints [-5.956, -49.496, 105.609, 215.565, 108.567, -180.049, -1180.02]
  MoveL 647 to (4.03, 195.62, 30) mm, rotated rx -90 ry -25 rz 54.24 deg; joints [-6.332, -49.606, 105.829, 215.332, 108.536, -179.801, -1174.238]
  MoveL 648 to (-1.12, 195.49, 20) mm, rotated rx -90 ry -25 rz 48.82 deg; joints [-6.709, -49.715, 106.043, 215.095, 108.501, -179.557, -1168.824]
  MoveL 649 to (-5.87, 195.78, 10) mm, rotated rx -90 ry -25 rz 43.82 deg; joints [-7.088, -49.822, 106.25, 214.856, 108.462, -179.315, -1163.823]
  MoveL 650 to (-10.16, 196.36, 0) mm, rotated rx -90 ry -25 rz 39.27 deg; joints [-7.468, -49.927, 106.451, 214.616, 108.422, -179.076, -1159.273]
  MoveL 651 to (28.22, 306.19, 290) mm, rotated rx -90 ry -25 rz -156.66 deg; joints [2.992, -46.023, 98.026, 220.579, 108.578, -187.075, -1323.337]
  Set speed (60.0 mm/s)
